	arModbusOdczytCykliczny[intPetlaPierwszySkan].bAdresUrzadzenia := bAdres;
	arModbusOdczytCykliczny[intPetlaPierwszySkan].bFunkcja := TO_BYTE(enumModbusKodyFunkcji.OdczytNRejestrow);
	arModbusOdczytCykliczny[intPetlaPierwszySkan].uiAdresRejestru := 50544;
	arModbusOdczytCykliczny[intPetlaPierwszySkan].ltCzestotliwosc := TIME_TO_LTIME(tMinimalnyCzasRaportowania);
	arModbusOdczytCykliczny[intPetlaPierwszySkan].pZmiennaReferencyjna := ADR(wMocCzynnaL1Hi);
	intPetlaPierwszySkan := intPetlaPierwszySkan + 1;
	
	arModbusOdczytCykliczny[intPetlaPierwszySkan].bAdresUrzadzenia := bAdres;
	arModbusOdczytCykliczny[intPetlaPierwszySkan].bFunkcja := TO_BYTE(enumModbusKodyFunkcji.OdczytNRejestrow);
	arModbusOdczytCykliczny[intPetlaPierwszySkan].uiAdresRejestru := 50545;
	arModbusOdczytCykliczny[intPetlaPierwszySkan].ltCzestotliwosc := TIME_TO_LTIME(tMinimalnyCzasRaportowania);
	arModbusOdczytCykliczny[intPetlaPierwszySkan].pZmiennaReferencyjna := ADR(wMocCzynnaL1Lo);
	intPetlaPierwszySkan := intPetlaPierwszySkan + 1;
	
	arModbusOdczytCykliczny[intPetlaPierwszySkan].bAdresUrzadzenia := bAdres;
	arModbusOdczytCykliczny[intPetlaPierwszySkan].bFunkcja := TO_BYTE(enumModbusKodyFunkcji.OdczytNRejestrow);
	arModbusOdczytCykliczny[intPetlaPierwszySkan].uiAdresRejestru := 50546;
	arModbusOdczytCykliczny[intPetlaPierwszySkan].ltCzestotliwosc := TIME_TO_LTIME(tMinimalnyCzasRaportowania);
	arModbusOdczytCykliczny[intPetlaPierwszySkan].pZmiennaReferencyjna := ADR(wMocCzynnaL2Hi);
	intPetlaPierwszySkan := intPetlaPierwszySkan + 1;
	
	arModbusOdczytCykliczny[intPetlaPierwszySkan].bAdresUrzadzenia := bAdres;
	arModbusOdczytCykliczny[intPetlaPierwszySkan].bFunkcja := TO_BYTE(enumModbusKodyFunkcji.OdczytNRejestrow);
	arModbusOdczytCykliczny[intPetlaPierwszySkan].uiAdresRejestru := 50547;
	arModbusOdczytCykliczny[intPetlaPierwszySkan].ltCzestotliwosc := TIME_TO_LTIME(tMinimalnyCzasRaportowania);
	arModbusOdczytCykliczny[intPetlaPierwszySkan].pZmiennaReferencyjna := ADR(wMocCzynnaL2Lo);
	intPetlaPierwszySkan := intPetlaPierwszySkan + 1;
	
	arModbusOdczytCykliczny[intPetlaPierwszySkan].bAdresUrzadzenia := bAdres;
	arModbusOdczytCykliczny[intPetlaPierwszySkan].bFunkcja := TO_BYTE(enumModbusKodyFunkcji.OdczytNRejestrow);
	arModbusOdczytCykliczny[intPetlaPierwszySkan].uiAdresRejestru := 50548;
	arModbusOdczytCykliczny[intPetlaPierwszySkan].ltCzestotliwosc := TIME_TO_LTIME(tMinimalnyCzasRaportowania);
	arModbusOdczytCykliczny[intPetlaPierwszySkan].pZmiennaReferencyjna := ADR(wMocCzynnaL3Hi);
	intPetlaPierwszySkan := intPetlaPierwszySkan + 1;
	
	arModbusOdczytCykliczny[intPetlaPierwszySkan].bAdresUrzadzenia := bAdres;
	arModbusOdczytCykliczny[intPetlaPierwszySkan].bFunkcja := TO_BYTE(enumModbusKodyFunkcji.OdczytNRejestrow);
	arModbusOdczytCykliczny[intPetlaPierwszySkan].uiAdresRejestru := 50549;
	arModbusOdczytCykliczny[intPetlaPierwszySkan].ltCzestotliwosc := TIME_TO_LTIME(tMinimalnyCzasRaportowania);
	arModbusOdczytCykliczny[intPetlaPierwszySkan].pZmiennaReferencyjna := ADR(wMocCzynnaL3Lo);
	intPetlaPierwszySkan := intPetlaPierwszySkan + 1;	
	
	arModbusOdczytCykliczny[intPetlaPierwszySkan].bAdresUrzadzenia := bAdres;
	arModbusOdczytCykliczny[intPetlaPierwszySkan].bFunkcja := TO_BYTE(enumModbusKodyFunkcji.OdczytNRejestrow);
	arModbusOdczytCykliczny[intPetlaPierwszySkan].uiAdresRejestru := 50556;
	arModbusOdczytCykliczny[intPetlaPierwszySkan].ltCzestotliwosc := TIME_TO_LTIME(tMinimalnyCzasRaportowania);
	arModbusOdczytCykliczny[intPetlaPierwszySkan].pZmiennaReferencyjna := ADR(wMocPozornaL1Hi);
	intPetlaPierwszySkan := intPetlaPierwszySkan + 1;

	arModbusOdczytCykliczny[intPetlaPierwszySkan].bAdresUrzadzenia := bAdres;
	arModbusOdczytCykliczny[intPetlaPierwszySkan].bFunkcja := TO_BYTE(enumModbusKodyFunkcji.OdczytNRejestrow);
	arModbusOdczytCykliczny[intPetlaPierwszySkan].uiAdresRejestru := 50557;
	arModbusOdczytCykliczny[intPetlaPierwszySkan].ltCzestotliwosc := TIME_TO_LTIME(tMinimalnyCzasRaportowania);
	arModbusOdczytCykliczny[intPetlaPierwszySkan].pZmiennaReferencyjna := ADR(wMocPozornaL1Lo);
	intPetlaPierwszySkan := intPetlaPierwszySkan + 1;	

	arModbusOdczytCykliczny[intPetlaPierwszySkan].bAdresUrzadzenia := bAdres;
	arModbusOdczytCykliczny[intPetlaPierwszySkan].bFunkcja := TO_BYTE(enumModbusKodyFunkcji.OdczytNRejestrow);
	arModbusOdczytCykliczny[intPetlaPierwszySkan].uiAdresRejestru := 50558;
	arModbusOdczytCykliczny[intPetlaPierwszySkan].ltCzestotliwosc := TIME_TO_LTIME(tMinimalnyCzasRaportowania);
	arModbusOdczytCykliczny[intPetlaPierwszySkan].pZmiennaReferencyjna := ADR(wMocPozornaL2Hi);
	intPetlaPierwszySkan := intPetlaPierwszySkan + 1;

	arModbusOdczytCykliczny[intPetlaPierwszySkan].bAdresUrzadzenia := bAdres;
	arModbusOdczytCykliczny[intPetlaPierwszySkan].bFunkcja := TO_BYTE(enumModbusKodyFunkcji.OdczytNRejestrow);
	arModbusOdczytCykliczny[intPetlaPierwszySkan].uiAdresRejestru := 50559;
	arModbusOdczytCykliczny[intPetlaPierwszySkan].ltCzestotliwosc := TIME_TO_LTIME(tMinimalnyCzasRaportowania);
	arModbusOdczytCykliczny[intPetlaPierwszySkan].pZmiennaReferencyjna := ADR(wMocPozornaL2Lo);
	intPetlaPierwszySkan := intPetlaPierwszySkan + 1;	

	arModbusOdczytCykliczny[intPetlaPierwszySkan].bAdresUrzadzenia := bAdres;
	arModbusOdczytCykliczny[intPetlaPierwszySkan].bFunkcja := TO_BYTE(enumModbusKodyFunkcji.OdczytNRejestrow);
	arModbusOdczytCykliczny[intPetlaPierwszySkan].uiAdresRejestru := 50560;
	arModbusOdczytCykliczny[intPetlaPierwszySkan].ltCzestotliwosc := TIME_TO_LTIME(tMinimalnyCzasRaportowania);
	arModbusOdczytCykliczny[intPetlaPierwszySkan].pZmiennaReferencyjna := ADR(wMocPozornaL3Hi);
	intPetlaPierwszySkan := intPetlaPierwszySkan + 1;

	arModbusOdczytCykliczny[intPetlaPierwszySkan].bAdresUrzadzenia := bAdres;
	arModbusOdczytCykliczny[intPetlaPierwszySkan].bFunkcja := TO_BYTE(enumModbusKodyFunkcji.OdczytNRejestrow);
	arModbusOdczytCykliczny[intPetlaPierwszySkan].uiAdresRejestru := 50561;
	arModbusOdczytCykliczny[intPetlaPierwszySkan].ltCzestotliwosc := TIME_TO_LTIME(tMinimalnyCzasRaportowania);
	arModbusOdczytCykliczny[intPetlaPierwszySkan].pZmiennaReferencyjna := ADR(wMocPozornaL3Lo);
	intPetlaPierwszySkan := intPetlaPierwszySkan + 1;	
	
	arModbusOdczytCykliczny[intPetlaPierwszySkan].bAdresUrzadzenia := bAdres;
	arModbusOdczytCykliczny[intPetlaPierwszySkan].bFunkcja := TO_BYTE(enumModbusKodyFunkcji.OdczytNRejestrow);
	arModbusOdczytCykliczny[intPetlaPierwszySkan].uiAdresRejestru := 50562;
	arModbusOdczytCykliczny[intPetlaPierwszySkan].ltCzestotliwosc := TIME_TO_LTIME(tMinimalnyCzasRaportowania);
	arModbusOdczytCykliczny[intPetlaPierwszySkan].pZmiennaReferencyjna := ADR(wWspolczynnikMocyL1Hi);
	intPetlaPierwszySkan := intPetlaPierwszySkan + 1;

	arModbusOdczytCykliczny[intPetlaPierwszySkan].bAdresUrzadzenia := bAdres;
	arModbusOdczytCykliczny[intPetlaPierwszySkan].bFunkcja := TO_BYTE(enumModbusKodyFunkcji.OdczytNRejestrow);
	arModbusOdczytCykliczny[intPetlaPierwszySkan].uiAdresRejestru := 50563;
	arModbusOdczytCykliczny[intPetlaPierwszySkan].ltCzestotliwosc := TIME_TO_LTIME(tMinimalnyCzasRaportowania);
	arModbusOdczytCykliczny[intPetlaPierwszySkan].pZmiennaReferencyjna := ADR(wWspolczynnikMocyL1Lo);
	intPetlaPierwszySkan := intPetlaPierwszySkan + 1;
	
	arModbusOdczytCykliczny[intPetlaPierwszySkan].bAdresUrzadzenia := bAdres;
	arModbusOdczytCykliczny[intPetlaPierwszySkan].bFunkcja := TO_BYTE(enumModbusKodyFunkcji.OdczytNRejestrow);
	arModbusOdczytCykliczny[intPetlaPierwszySkan].uiAdresRejestru := 50564;
	arModbusOdczytCykliczny[intPetlaPierwszySkan].ltCzestotliwosc := TIME_TO_LTIME(tMinimalnyCzasRaportowania);
	arModbusOdczytCykliczny[intPetlaPierwszySkan].pZmiennaReferencyjna := ADR(wWspolczynnikMocyL2Hi);
	intPetlaPierwszySkan := intPetlaPierwszySkan + 1;

	arModbusOdczytCykliczny[intPetlaPierwszySkan].bAdresUrzadzenia := bAdres;
	arModbusOdczytCykliczny[intPetlaPierwszySkan].bFunkcja := TO_BYTE(enumModbusKodyFunkcji.OdczytNRejestrow);
	arModbusOdczytCykliczny[intPetlaPierwszySkan].uiAdresRejestru := 50565;
	arModbusOdczytCykliczny[intPetlaPierwszySkan].ltCzestotliwosc := TIME_TO_LTIME(tMinimalnyCzasRaportowania);
	arModbusOdczytCykliczny[intPetlaPierwszySkan].pZmiennaReferencyjna := ADR(wWspolczynnikMocyL2Lo);
	intPetlaPierwszySkan := intPetlaPierwszySkan + 1;
	
	arModbusOdczytCykliczny[intPetlaPierwszySkan].bAdresUrzadzenia := bAdres;
	arModbusOdczytCykliczny[intPetlaPierwszySkan].bFunkcja := TO_BYTE(enumModbusKodyFunkcji.OdczytNRejestrow);
	arModbusOdczytCykliczny[intPetlaPierwszySkan].uiAdresRejestru := 50566;
	arModbusOdczytCykliczny[intPetlaPierwszySkan].ltCzestotliwosc := TIME_TO_LTIME(tMinimalnyCzasRaportowania);
	arModbusOdczytCykliczny[intPetlaPierwszySkan].pZmiennaReferencyjna := ADR(wWspolczynnikMocyL3Hi);
	intPetlaPierwszySkan := intPetlaPierwszySkan + 1;

	arModbusOdczytCykliczny[intPetlaPierwszySkan].bAdresUrzadzenia := bAdres;
	arModbusOdczytCykliczny[intPetlaPierwszySkan].bFunkcja := TO_BYTE(enumModbusKodyFunkcji.OdczytNRejestrow);
	arModbusOdczytCykliczny[intPetlaPierwszySkan].uiAdresRejestru := 50567;
	arModbusOdczytCykliczny[intPetlaPierwszySkan].ltCzestotliwosc := TIME_TO_LTIME(tMinimalnyCzasRaportowania);
	arModbusOdczytCykliczny[intPetlaPierwszySkan].pZmiennaReferencyjna := ADR(wWspolczynnikMocyL3Lo);
	intPetlaPierwszySkan := intPetlaPierwszySkan + 1;
	
	arModbusOdczytCykliczny[intPetlaPierwszySkan].bAdresUrzadzenia := bAdres;
	arModbusOdczytCykliczny[intPetlaPierwszySkan].bFunkcja := TO_BYTE(enumModbusKodyFunkcji.OdczytNRejestrow);
	arModbusOdczytCykliczny[intPetlaPierwszySkan].uiAdresRejestru := 856;
	arModbusOdczytCykliczny[intPetlaPierwszySkan].ltCzestotliwosc := TIME_TO_LTIME(tMinimalnyCzasRaportowania);
	arModbusOdczytCykliczny[intPetlaPierwszySkan].pZmiennaReferencyjna := ADR(wEnergiaCzynnaPobranaHi);
	intPetlaPierwszySkan := intPetlaPierwszySkan + 1;

	arModbusOdczytCykliczny[intPetlaPierwszySkan].bAdresUrzadzenia := bAdres;
	arModbusOdczytCykliczny[intPetlaPierwszySkan].bFunkcja := TO_BYTE(enumModbusKodyFunkcji.OdczytNRejestrow);
	arModbusOdczytCykliczny[intPetlaPierwszySkan].uiAdresRejestru := 857;
	arModbusOdczytCykliczny[intPetlaPierwszySkan].ltCzestotliwosc := TIME_TO_LTIME(tMinimalnyCzasRaportowania);
	arModbusOdczytCykliczny[intPetlaPierwszySkan].pZmiennaReferencyjna := ADR(wEnergiaCzynnaPobranaLo);
	intPetlaPierwszySkan := intPetlaPierwszySkan + 1;
	
	arModbusOdczytCykliczny[intPetlaPierwszySkan].bAdresUrzadzenia := bAdres;
	arModbusOdczytCykliczny[intPetlaPierwszySkan].bFunkcja := TO_BYTE(enumModbusKodyFunkcji.OdczytNRejestrow);
	arModbusOdczytCykliczny[intPetlaPierwszySkan].uiAdresRejestru := 858;
	arModbusOdczytCykliczny[intPetlaPierwszySkan].ltCzestotliwosc := TIME_TO_LTIME(tMinimalnyCzasRaportowania);
	arModbusOdczytCykliczny[intPetlaPierwszySkan].pZmiennaReferencyjna := ADR(wEnergiaBiernaPobranaHi);
	intPetlaPierwszySkan := intPetlaPierwszySkan + 1;

	arModbusOdczytCykliczny[intPetlaPierwszySkan].bAdresUrzadzenia := bAdres;
	arModbusOdczytCykliczny[intPetlaPierwszySkan].bFunkcja := TO_BYTE(enumModbusKodyFunkcji.OdczytNRejestrow);
	arModbusOdczytCykliczny[intPetlaPierwszySkan].uiAdresRejestru := 859;
	arModbusOdczytCykliczny[intPetlaPierwszySkan].ltCzestotliwosc := TIME_TO_LTIME(tMinimalnyCzasRaportowania);
	arModbusOdczytCykliczny[intPetlaPierwszySkan].pZmiennaReferencyjna := ADR(wEnergiaBiernaPobranaLo);
	intPetlaPierwszySkan := intPetlaPierwszySkan + 1;
	
	arModbusOdczytCykliczny[intPetlaPierwszySkan].bAdresUrzadzenia := bAdres;
	arModbusOdczytCykliczny[intPetlaPierwszySkan].bFunkcja := TO_BYTE(enumModbusKodyFunkcji.OdczytNRejestrow);
	arModbusOdczytCykliczny[intPetlaPierwszySkan].uiAdresRejestru := 860;
	arModbusOdczytCykliczny[intPetlaPierwszySkan].ltCzestotliwosc := TIME_TO_LTIME(tMinimalnyCzasRaportowania);
	arModbusOdczytCykliczny[intPetlaPierwszySkan].pZmiennaReferencyjna := ADR(wEnergiaPozornaPobranaHi);
	intPetlaPierwszySkan := intPetlaPierwszySkan + 1;

	arModbusOdczytCykliczny[intPetlaPierwszySkan].bAdresUrzadzenia := bAdres;
	arModbusOdczytCykliczny[intPetlaPierwszySkan].bFunkcja := TO_BYTE(enumModbusKodyFunkcji.OdczytNRejestrow);
	arModbusOdczytCykliczny[intPetlaPierwszySkan].uiAdresRejestru := 861;
	arModbusOdczytCykliczny[intPetlaPierwszySkan].ltCzestotliwosc := TIME_TO_LTIME(tMinimalnyCzasRaportowania);
	arModbusOdczytCykliczny[intPetlaPierwszySkan].pZmiennaReferencyjna := ADR(wEnergiaPozornaPobranaLo);
	intPetlaPierwszySkan := intPetlaPierwszySkan + 1;
	
	arModbusOdczytCykliczny[intPetlaPierwszySkan].bAdresUrzadzenia := bAdres;
	arModbusOdczytCykliczny[intPetlaPierwszySkan].bFunkcja := TO_BYTE(enumModbusKodyFunkcji.OdczytNRejestrow);
	arModbusOdczytCykliczny[intPetlaPierwszySkan].uiAdresRejestru := 51038;
	arModbusOdczytCykliczny[intPetlaPierwszySkan].ltCzestotliwosc := TIME_TO_LTIME(tMinimalnyCzasRaportowania);
	arModbusOdczytCykliczny[intPetlaPierwszySkan].pZmiennaReferencyjna := ADR(wPradSredniL1Hi);
	intPetlaPierwszySkan := intPetlaPierwszySkan + 1;

	arModbusOdczytCykliczny[intPetlaPierwszySkan].bAdresUrzadzenia := bAdres;
	arModbusOdczytCykliczny[intPetlaPierwszySkan].bFunkcja := TO_BYTE(enumModbusKodyFunkcji.OdczytNRejestrow);
	arModbusOdczytCykliczny[intPetlaPierwszySkan].uiAdresRejestru := 51039;
	arModbusOdczytCykliczny[intPetlaPierwszySkan].ltCzestotliwosc := TIME_TO_LTIME(tMinimalnyCzasRaportowania);
	arModbusOdczytCykliczny[intPetlaPierwszySkan].pZmiennaReferencyjna := ADR(wPradSredniL1Lo);
	intPetlaPierwszySkan := intPetlaPierwszySkan + 1;
	
	arModbusOdczytCykliczny[intPetlaPierwszySkan].bAdresUrzadzenia := bAdres;
	arModbusOdczytCykliczny[intPetlaPierwszySkan].bFunkcja := TO_BYTE(enumModbusKodyFunkcji.OdczytNRejestrow);
	arModbusOdczytCykliczny[intPetlaPierwszySkan].uiAdresRejestru := 51040;
	arModbusOdczytCykliczny[intPetlaPierwszySkan].ltCzestotliwosc := TIME_TO_LTIME(tMinimalnyCzasRaportowania);
	arModbusOdczytCykliczny[intPetlaPierwszySkan].pZmiennaReferencyjna := ADR(wPradSredniL2Hi);
	intPetlaPierwszySkan := intPetlaPierwszySkan + 1;

	arModbusOdczytCykliczny[intPetlaPierwszySkan].bAdresUrzadzenia := bAdres;
	arModbusOdczytCykliczny[intPetlaPierwszySkan].bFunkcja := TO_BYTE(enumModbusKodyFunkcji.OdczytNRejestrow);
	arModbusOdczytCykliczny[intPetlaPierwszySkan].uiAdresRejestru := 51041;
	arModbusOdczytCykliczny[intPetlaPierwszySkan].ltCzestotliwosc := TIME_TO_LTIME(tMinimalnyCzasRaportowania);
	arModbusOdczytCykliczny[intPetlaPierwszySkan].pZmiennaReferencyjna := ADR(wPradSredniL2Lo);
	intPetlaPierwszySkan := intPetlaPierwszySkan + 1;
	
	arModbusOdczytCykliczny[intPetlaPierwszySkan].bAdresUrzadzenia := bAdres;
	arModbusOdczytCykliczny[intPetlaPierwszySkan].bFunkcja := TO_BYTE(enumModbusKodyFunkcji.OdczytNRejestrow);
	arModbusOdczytCykliczny[intPetlaPierwszySkan].uiAdresRejestru := 51042;
	arModbusOdczytCykliczny[intPetlaPierwszySkan].ltCzestotliwosc := TIME_TO_LTIME(tMinimalnyCzasRaportowania);
	arModbusOdczytCykliczny[intPetlaPierwszySkan].pZmiennaReferencyjna := ADR(wPradSredniL3Hi);
	intPetlaPierwszySkan := intPetlaPierwszySkan + 1;

	arModbusOdczytCykliczny[intPetlaPierwszySkan].bAdresUrzadzenia := bAdres;
	arModbusOdczytCykliczny[intPetlaPierwszySkan].bFunkcja := TO_BYTE(enumModbusKodyFunkcji.OdczytNRejestrow);
	arModbusOdczytCykliczny[intPetlaPierwszySkan].uiAdresRejestru := 51043;
	arModbusOdczytCykliczny[intPetlaPierwszySkan].ltCzestotliwosc := TIME_TO_LTIME(tMinimalnyCzasRaportowania);
	arModbusOdczytCykliczny[intPetlaPierwszySkan].pZmiennaReferencyjna := ADR(wPradSredniL3Lo);
	intPetlaPierwszySkan := intPetlaPierwszySkan + 1;

	arModbusOdczytCykliczny[intPetlaPierwszySkan].bAdresUrzadzenia := bAdres;
	arModbusOdczytCykliczny[intPetlaPierwszySkan].bFunkcja := TO_BYTE(enumModbusKodyFunkcji.OdczytNRejestrow);
	arModbusOdczytCykliczny[intPetlaPierwszySkan].uiAdresRejestru := 51046;
	arModbusOdczytCykliczny[intPetlaPierwszySkan].ltCzestotliwosc := TIME_TO_LTIME(tMinimalnyCzasRaportowania);
	arModbusOdczytCykliczny[intPetlaPierwszySkan].pZmiennaReferencyjna := ADR(wMocCzynnaSredniaHi);
	intPetlaPierwszySkan := intPetlaPierwszySkan + 1;

	arModbusOdczytCykliczny[intPetlaPierwszySkan].bAdresUrzadzenia := bAdres;
	arModbusOdczytCykliczny[intPetlaPierwszySkan].bFunkcja := TO_BYTE(enumModbusKodyFunkcji.OdczytNRejestrow);
	arModbusOdczytCykliczny[intPetlaPierwszySkan].uiAdresRejestru := 51047;
	arModbusOdczytCykliczny[intPetlaPierwszySkan].ltCzestotliwosc := TIME_TO_LTIME(tMinimalnyCzasRaportowania);
	arModbusOdczytCykliczny[intPetlaPierwszySkan].pZmiennaReferencyjna := ADR(wMocCzynnaSredniaLo);
	intPetlaPierwszySkan := intPetlaPierwszySkan + 1;

	arModbusOdczytCykliczny[intPetlaPierwszySkan].bAdresUrzadzenia := bAdres;
	arModbusOdczytCykliczny[intPetlaPierwszySkan].bFunkcja := TO_BYTE(enumModbusKodyFunkcji.OdczytNRejestrow);
	arModbusOdczytCykliczny[intPetlaPierwszySkan].uiAdresRejestru := 51052;
	arModbusOdczytCykliczny[intPetlaPierwszySkan].ltCzestotliwosc := TIME_TO_LTIME(tMinimalnyCzasRaportowania);
	arModbusOdczytCykliczny[intPetlaPierwszySkan].pZmiennaReferencyjna := ADR(wMocBiernaSredniaHi);
	intPetlaPierwszySkan := intPetlaPierwszySkan + 1;

	arModbusOdczytCykliczny[intPetlaPierwszySkan].bAdresUrzadzenia := bAdres;
	arModbusOdczytCykliczny[intPetlaPierwszySkan].bFunkcja := TO_BYTE(enumModbusKodyFunkcji.OdczytNRejestrow);
	arModbusOdczytCykliczny[intPetlaPierwszySkan].uiAdresRejestru := 51053;
	arModbusOdczytCykliczny[intPetlaPierwszySkan].ltCzestotliwosc := TIME_TO_LTIME(tMinimalnyCzasRaportowania);
	arModbusOdczytCykliczny[intPetlaPierwszySkan].pZmiennaReferencyjna := ADR(wMocBiernaSredniaLo);
	intPetlaPierwszySkan := intPetlaPierwszySkan + 1;

	arModbusOdczytCykliczny[intPetlaPierwszySkan].bAdresUrzadzenia := bAdres;
	arModbusOdczytCykliczny[intPetlaPierwszySkan].bFunkcja := TO_BYTE(enumModbusKodyFunkcji.OdczytNRejestrow);
	arModbusOdczytCykliczny[intPetlaPierwszySkan].uiAdresRejestru := 51054;
	arModbusOdczytCykliczny[intPetlaPierwszySkan].ltCzestotliwosc := TIME_TO_LTIME(tMinimalnyCzasRaportowania);
	arModbusOdczytCykliczny[intPetlaPierwszySkan].pZmiennaReferencyjna := ADR(wMocPozornaSredniaHi);
	intPetlaPierwszySkan := intPetlaPierwszySkan + 1;

	arModbusOdczytCykliczny[intPetlaPierwszySkan].bAdresUrzadzenia := bAdres;
	arModbusOdczytCykliczny[intPetlaPierwszySkan].bFunkcja := TO_BYTE(enumModbusKodyFunkcji.OdczytNRejestrow);
	arModbusOdczytCykliczny[intPetlaPierwszySkan].uiAdresRejestru := 51055;
	arModbusOdczytCykliczny[intPetlaPierwszySkan].ltCzestotliwosc := TIME_TO_LTIME(tMinimalnyCzasRaportowania);
	arModbusOdczytCykliczny[intPetlaPierwszySkan].pZmiennaReferencyjna := ADR(wMocPozornaSredniaLo);
	intPetlaPierwszySkan := intPetlaPierwszySkan + 1;

	arModbusOdczytCykliczny[intPetlaPierwszySkan].bAdresUrzadzenia := bAdres;
	arModbusOdczytCykliczny[intPetlaPierwszySkan].bFunkcja := TO_BYTE(enumModbusKodyFunkcji.OdczytNRejestrow);
	arModbusOdczytCykliczny[intPetlaPierwszySkan].uiAdresRejestru := 51062;
	arModbusOdczytCykliczny[intPetlaPierwszySkan].ltCzestotliwosc := TIME_TO_LTIME(tMinimalnyCzasRaportowania);
	arModbusOdczytCykliczny[intPetlaPierwszySkan].pZmiennaReferencyjna := ADR(wMaksymalneNapiecieL1Hi);
	intPetlaPierwszySkan := intPetlaPierwszySkan + 1;

	arModbusOdczytCykliczny[intPetlaPierwszySkan].bAdresUrzadzenia := bAdres;
	arModbusOdczytCykliczny[intPetlaPierwszySkan].bFunkcja := TO_BYTE(enumModbusKodyFunkcji.OdczytNRejestrow);
	arModbusOdczytCykliczny[intPetlaPierwszySkan].uiAdresRejestru := 51063;
	arModbusOdczytCykliczny[intPetlaPierwszySkan].ltCzestotliwosc := TIME_TO_LTIME(tMinimalnyCzasRaportowania);
	arModbusOdczytCykliczny[intPetlaPierwszySkan].pZmiennaReferencyjna := ADR(wMaksymalneNapiecieL1Lo);
	intPetlaPierwszySkan := intPetlaPierwszySkan + 1;

	arModbusOdczytCykliczny[intPetlaPierwszySkan].bAdresUrzadzenia := bAdres;
	arModbusOdczytCykliczny[intPetlaPierwszySkan].bFunkcja := TO_BYTE(enumModbusKodyFunkcji.OdczytNRejestrow);
	arModbusOdczytCykliczny[intPetlaPierwszySkan].uiAdresRejestru := 51064;
	arModbusOdczytCykliczny[intPetlaPierwszySkan].ltCzestotliwosc := TIME_TO_LTIME(tMinimalnyCzasRaportowania);
	arModbusOdczytCykliczny[intPetlaPierwszySkan].pZmiennaReferencyjna := ADR(wMaksymalneNapiecieL2Hi);
	intPetlaPierwszySkan := intPetlaPierwszySkan + 1;

	arModbusOdczytCykliczny[intPetlaPierwszySkan].bAdresUrzadzenia := bAdres;
	arModbusOdczytCykliczny[intPetlaPierwszySkan].bFunkcja := TO_BYTE(enumModbusKodyFunkcji.OdczytNRejestrow);
	arModbusOdczytCykliczny[intPetlaPierwszySkan].uiAdresRejestru := 51065;
	arModbusOdczytCykliczny[intPetlaPierwszySkan].ltCzestotliwosc := TIME_TO_LTIME(tMinimalnyCzasRaportowania);
	arModbusOdczytCykliczny[intPetlaPierwszySkan].pZmiennaReferencyjna := ADR(wMaksymalneNapiecieL2Lo);
	intPetlaPierwszySkan := intPetlaPierwszySkan + 1;

	arModbusOdczytCykliczny[intPetlaPierwszySkan].bAdresUrzadzenia := bAdres;
	arModbusOdczytCykliczny[intPetlaPierwszySkan].bFunkcja := TO_BYTE(enumModbusKodyFunkcji.OdczytNRejestrow);
	arModbusOdczytCykliczny[intPetlaPierwszySkan].uiAdresRejestru := 51066;
	arModbusOdczytCykliczny[intPetlaPierwszySkan].ltCzestotliwosc := TIME_TO_LTIME(tMinimalnyCzasRaportowania);
	arModbusOdczytCykliczny[intPetlaPierwszySkan].pZmiennaReferencyjna := ADR(wMaksymalneNapiecieL3Hi);
	intPetlaPierwszySkan := intPetlaPierwszySkan + 1;

	arModbusOdczytCykliczny[intPetlaPierwszySkan].bAdresUrzadzenia := bAdres;
	arModbusOdczytCykliczny[intPetlaPierwszySkan].bFunkcja := TO_BYTE(enumModbusKodyFunkcji.OdczytNRejestrow);
	arModbusOdczytCykliczny[intPetlaPierwszySkan].uiAdresRejestru := 51067;
	arModbusOdczytCykliczny[intPetlaPierwszySkan].ltCzestotliwosc := TIME_TO_LTIME(tMinimalnyCzasRaportowania);
	arModbusOdczytCykliczny[intPetlaPierwszySkan].pZmiennaReferencyjna := ADR(wMaksymalneNapiecieL3Lo);
	intPetlaPierwszySkan := intPetlaPierwszySkan + 1;

	arModbusOdczytCykliczny[intPetlaPierwszySkan].bAdresUrzadzenia := bAdres;
	arModbusOdczytCykliczny[intPetlaPierwszySkan].bFunkcja := TO_BYTE(enumModbusKodyFunkcji.OdczytNRejestrow);
	arModbusOdczytCykliczny[intPetlaPierwszySkan].uiAdresRejestru := 51539;
	arModbusOdczytCykliczny[intPetlaPierwszySkan].ltCzestotliwosc := TIME_TO_LTIME(tMinimalnyCzasRaportowania);
	arModbusOdczytCykliczny[intPetlaPierwszySkan].pZmiennaReferencyjna := ADR(wTHDNapieciaL1);
	intPetlaPierwszySkan := intPetlaPierwszySkan + 1;

	arModbusOdczytCykliczny[intPetlaPierwszySkan].bAdresUrzadzenia := bAdres;
	arModbusOdczytCykliczny[intPetlaPierwszySkan].bFunkcja := TO_BYTE(enumModbusKodyFunkcji.OdczytNRejestrow);
	arModbusOdczytCykliczny[intPetlaPierwszySkan].uiAdresRejestru := 51540;
	arModbusOdczytCykliczny[intPetlaPierwszySkan].ltCzestotliwosc := TIME_TO_LTIME(tMinimalnyCzasRaportowania);
	arModbusOdczytCykliczny[intPetlaPierwszySkan].pZmiennaReferencyjna := ADR(wTHDNapieciaL2);
	intPetlaPierwszySkan := intPetlaPierwszySkan + 1;

	arModbusOdczytCykliczny[intPetlaPierwszySkan].bAdresUrzadzenia := bAdres;
	arModbusOdczytCykliczny[intPetlaPierwszySkan].bFunkcja := TO_BYTE(enumModbusKodyFunkcji.OdczytNRejestrow);
	arModbusOdczytCykliczny[intPetlaPierwszySkan].uiAdresRejestru := 51541;
	arModbusOdczytCykliczny[intPetlaPierwszySkan].ltCzestotliwosc := TIME_TO_LTIME(tMinimalnyCzasRaportowania);
	arModbusOdczytCykliczny[intPetlaPierwszySkan].pZmiennaReferencyjna := ADR(wTHDNapieciaL3);
	intPetlaPierwszySkan := intPetlaPierwszySkan + 1;

	arModbusOdczytCykliczny[intPetlaPierwszySkan].bAdresUrzadzenia := bAdres;
	arModbusOdczytCykliczny[intPetlaPierwszySkan].bFunkcja := TO_BYTE(enumModbusKodyFunkcji.OdczytNRejestrow);
	arModbusOdczytCykliczny[intPetlaPierwszySkan].uiAdresRejestru := 51542;
	arModbusOdczytCykliczny[intPetlaPierwszySkan].ltCzestotliwosc := TIME_TO_LTIME(tMinimalnyCzasRaportowania);
	arModbusOdczytCykliczny[intPetlaPierwszySkan].pZmiennaReferencyjna := ADR(wTHDPraduL1);
	intPetlaPierwszySkan := intPetlaPierwszySkan + 1;

	arModbusOdczytCykliczny[intPetlaPierwszySkan].bAdresUrzadzenia := bAdres;
	arModbusOdczytCykliczny[intPetlaPierwszySkan].bFunkcja := TO_BYTE(enumModbusKodyFunkcji.OdczytNRejestrow);
	arModbusOdczytCykliczny[intPetlaPierwszySkan].uiAdresRejestru := 51543;
	arModbusOdczytCykliczny[intPetlaPierwszySkan].ltCzestotliwosc := TIME_TO_LTIME(tMinimalnyCzasRaportowania);
	arModbusOdczytCykliczny[intPetlaPierwszySkan].pZmiennaReferencyjna := ADR(wTHDPraduL2);
	intPetlaPierwszySkan := intPetlaPierwszySkan + 1;

	arModbusOdczytCykliczny[intPetlaPierwszySkan].bAdresUrzadzenia := bAdres;
	arModbusOdczytCykliczny[intPetlaPierwszySkan].bFunkcja := TO_BYTE(enumModbusKodyFunkcji.OdczytNRejestrow);
	arModbusOdczytCykliczny[intPetlaPierwszySkan].uiAdresRejestru := 51544;
	arModbusOdczytCykliczny[intPetlaPierwszySkan].ltCzestotliwosc := TIME_TO_LTIME(tMinimalnyCzasRaportowania);
	arModbusOdczytCykliczny[intPetlaPierwszySkan].pZmiennaReferencyjna := ADR(wTHDPraduL3);
	intPetlaPierwszySkan := intPetlaPierwszySkan + 1;
END_IF

//obsluga komunikatu przychodzacego z IZE

IF 	sKomunikat <> sKomunikatPamiec AND xPoInicjalizacji THEN
	sKomunikatPamiec := sKomunikat;
	IF fnIDOdbiorcyMatch(sKomunikat , sIdInstancji) THEN
		sDane := '';
		//zapytanie typu Q
		IF fnKomunikatTyp(sKomunikat) = 'Q' AND arModbusStatusKomunikacji[bAdres] = enumModbusStatus.KomunikacjaPrawidlowa THEN
			//Napięcia fazowe
			IF fnKomunikatDaneSzukajWartosci(sKomunikat , 'VOLTL1=') = '?' OR fnKomunikatDaneSzukajWartosci(sKomunikat , 'ALL=') = '?' THEN
				fnKomunikatDaneDodaj_xOverFlow(sDane := sDane , sAtrybut := 'VOLTL1=' , sWartosc := REAL_TO_STRING(rNapiecieL1) , xOverFlow := xOverFlow);
				IF xOverFlow = TRUE THEN
					fnZapiszKomunikat(	sCalyKomunikat := '' ,
								sTypKomunikatu := 'A' ,
								sMnemonik := sMnemonik ,
								sMACAdres := sMACAdres ,
								sIDNadawcy := sIdInstancji ,
								sIDOdbiorcy := sIdAplikacji ,
								sDaneZapasowe := sDaneZapasowe ,
								sDane := sDane ,
								arTablicaKomunikatow := arTablicaKomunikatow ,
								intTablicaKomunikatowZnacznikZapisu := intTablicaKomunikatowZnacznikZapisu ,
								intTablicaKomunikatowRozmiar := intTablicaKomunikatowRozmiar ,
								sWyslanyKomunikat := sWyslanyKomunikatDummy);
					sDane := '';
				END_IF
			END_IF
			IF fnKomunikatDaneSzukajWartosci(sKomunikat , 'VOLTL2=') = '?' OR fnKomunikatDaneSzukajWartosci(sKomunikat , 'ALL=') = '?' THEN
				fnKomunikatDaneDodaj_xOverFlow(sDane := sDane , sAtrybut := 'VOLTL2=' , sWartosc := REAL_TO_STRING(rNapiecieL2) , xOverFlow := xOverFlow);
				IF xOverFlow = TRUE THEN
					fnZapiszKomunikat(	sCalyKomunikat := '' ,
								sTypKomunikatu := 'A' ,
								sMnemonik := sMnemonik ,
								sMACAdres := sMACAdres ,
								sIDNadawcy := sIdInstancji ,
								sIDOdbiorcy := sIdAplikacji ,
								sDaneZapasowe := sDaneZapasowe ,
								sDane := sDane ,
								arTablicaKomunikatow := arTablicaKomunikatow ,
								intTablicaKomunikatowZnacznikZapisu := intTablicaKomunikatowZnacznikZapisu ,
								intTablicaKomunikatowRozmiar := intTablicaKomunikatowRozmiar ,
								sWyslanyKomunikat := sWyslanyKomunikatDummy);
					sDane := '';
				END_IF	
			END_IF	
			IF fnKomunikatDaneSzukajWartosci(sKomunikat , 'VOLTL3=') = '?' OR fnKomunikatDaneSzukajWartosci(sKomunikat , 'ALL=') = '?' THEN
				fnKomunikatDaneDodaj_xOverFlow(sDane := sDane , sAtrybut := 'VOLTL3=' , sWartosc := REAL_TO_STRING(rNapiecieL3) , xOverFlow := xOverFlow);	
				IF xOverFlow = TRUE THEN
					fnZapiszKomunikat(	sCalyKomunikat := '' ,
								sTypKomunikatu := 'A' ,
								sMnemonik := sMnemonik ,
								sMACAdres := sMACAdres ,
								sIDNadawcy := sIdInstancji ,
								sIDOdbiorcy := sIdAplikacji ,
								sDaneZapasowe := sDaneZapasowe ,
								sDane := sDane ,
								arTablicaKomunikatow := arTablicaKomunikatow ,
								intTablicaKomunikatowZnacznikZapisu := intTablicaKomunikatowZnacznikZapisu ,
								intTablicaKomunikatowRozmiar := intTablicaKomunikatowRozmiar ,
								sWyslanyKomunikat := sWyslanyKomunikatDummy);
					sDane := '';
				END_IF	
			END_IF
			//Napięcia przewodowe
			IF fnKomunikatDaneSzukajWartosci(sKomunikat , 'VOLTL1L2=') = '?' OR fnKomunikatDaneSzukajWartosci(sKomunikat , 'ALL=') = '?' THEN
				fnKomunikatDaneDodaj_xOverFlow(sDane := sDane , sAtrybut := 'VOLTL1L2=' , sWartosc := REAL_TO_STRING(rNapiecieL1L2) , xOverFlow := xOverFlow);	
				IF xOverFlow = TRUE THEN
					fnZapiszKomunikat(	sCalyKomunikat := '' ,
								sTypKomunikatu := 'A' ,
								sMnemonik := sMnemonik ,
								sMACAdres := sMACAdres ,
								sIDNadawcy := sIdInstancji ,
								sIDOdbiorcy := sIdAplikacji ,
								sDaneZapasowe := sDaneZapasowe ,
								sDane := sDane ,
								arTablicaKomunikatow := arTablicaKomunikatow ,
								intTablicaKomunikatowZnacznikZapisu := intTablicaKomunikatowZnacznikZapisu ,
								intTablicaKomunikatowRozmiar := intTablicaKomunikatowRozmiar ,
								sWyslanyKomunikat := sWyslanyKomunikatDummy);
					sDane := '';
				END_IF	
			END_IF
			IF fnKomunikatDaneSzukajWartosci(sKomunikat , 'VOLTL2L3=') = '?' OR fnKomunikatDaneSzukajWartosci(sKomunikat , 'ALL=') = '?' THEN
				fnKomunikatDaneDodaj_xOverFlow(sDane := sDane , sAtrybut := 'VOLTL2L3=' , sWartosc := REAL_TO_STRING(rNapiecieL2L3) , xOverFlow := xOverFlow);	
				IF xOverFlow = TRUE THEN
					fnZapiszKomunikat(	sCalyKomunikat := '' ,
								sTypKomunikatu := 'A' ,
								sMnemonik := sMnemonik ,
								sMACAdres := sMACAdres ,
								sIDNadawcy := sIdInstancji ,
								sIDOdbiorcy := sIdAplikacji ,
								sDaneZapasowe := sDaneZapasowe ,
								sDane := sDane ,
								arTablicaKomunikatow := arTablicaKomunikatow ,
								intTablicaKomunikatowZnacznikZapisu := intTablicaKomunikatowZnacznikZapisu ,
								intTablicaKomunikatowRozmiar := intTablicaKomunikatowRozmiar ,
								sWyslanyKomunikat := sWyslanyKomunikatDummy);
					sDane := '';
				END_IF	
			END_IF	
			IF fnKomunikatDaneSzukajWartosci(sKomunikat , 'VOLTL3L1=') = '?' OR fnKomunikatDaneSzukajWartosci(sKomunikat , 'ALL=') = '?' THEN
				fnKomunikatDaneDodaj_xOverFlow(sDane := sDane , sAtrybut := 'VOLTL3L1=' , sWartosc := REAL_TO_STRING(rNapiecieL3L1) , xOverFlow := xOverFlow);	
				IF xOverFlow = TRUE THEN
					fnZapiszKomunikat(	sCalyKomunikat := '' ,
								sTypKomunikatu := 'A' ,
								sMnemonik := sMnemonik ,
								sMACAdres := sMACAdres ,
								sIDNadawcy := sIdInstancji ,
								sIDOdbiorcy := sIdAplikacji ,
								sDaneZapasowe := sDaneZapasowe ,
								sDane := sDane ,
								arTablicaKomunikatow := arTablicaKomunikatow ,
								intTablicaKomunikatowZnacznikZapisu := intTablicaKomunikatowZnacznikZapisu ,
								intTablicaKomunikatowRozmiar := intTablicaKomunikatowRozmiar ,
								sWyslanyKomunikat := sWyslanyKomunikatDummy);
					sDane := '';
				END_IF	
			END_IF
			//Częstotliwość 
			IF fnKomunikatDaneSzukajWartosci(sKomunikat , 'CZEST=') = '?' OR fnKomunikatDaneSzukajWartosci(sKomunikat , 'ALL=') = '?' THEN
				fnKomunikatDaneDodaj_xOverFlow(sDane := sDane , sAtrybut := 'CZEST=' , sWartosc := REAL_TO_STRING(rCzestotliwosc) , xOverFlow := xOverFlow);	
				IF xOverFlow = TRUE THEN
					fnZapiszKomunikat(	sCalyKomunikat := '' ,
								sTypKomunikatu := 'A' ,
								sMnemonik := sMnemonik ,
								sMACAdres := sMACAdres ,
								sIDNadawcy := sIdInstancji ,
								sIDOdbiorcy := sIdAplikacji ,
								sDaneZapasowe := sDaneZapasowe ,
								sDane := sDane ,
								arTablicaKomunikatow := arTablicaKomunikatow ,
								intTablicaKomunikatowZnacznikZapisu := intTablicaKomunikatowZnacznikZapisu ,
								intTablicaKomunikatowRozmiar := intTablicaKomunikatowRozmiar ,
								sWyslanyKomunikat := sWyslanyKomunikatDummy);
					sDane := '';
				END_IF	
			END_IF
			//Czas pracy 
			IF fnKomunikatDaneSzukajWartosci(sKomunikat , 'CZAS=') = '?' OR fnKomunikatDaneSzukajWartosci(sKomunikat , 'ALL=') = '?' THEN
				fnKomunikatDaneDodaj_xOverFlow(sDane := sDane , sAtrybut := 'CZAS=' , sWartosc := REAL_TO_STRING(rCzasPracyAnalizatora) , xOverFlow := xOverFlow);	
				IF xOverFlow = TRUE THEN
					fnZapiszKomunikat(	sCalyKomunikat := '' ,
								sTypKomunikatu := 'A' ,
								sMnemonik := sMnemonik ,
								sMACAdres := sMACAdres ,
								sIDNadawcy := sIdInstancji ,
								sIDOdbiorcy := sIdAplikacji ,
								sDaneZapasowe := sDaneZapasowe ,
								sDane := sDane ,
								arTablicaKomunikatow := arTablicaKomunikatow ,
								intTablicaKomunikatowZnacznikZapisu := intTablicaKomunikatowZnacznikZapisu ,
								intTablicaKomunikatowRozmiar := intTablicaKomunikatowRozmiar ,
								sWyslanyKomunikat := sWyslanyKomunikatDummy);
					sDane := '';
				END_IF	
			END_IF
			//Prądy fazowe
			IF fnKomunikatDaneSzukajWartosci(sKomunikat , 'AMPERL1=') = '?' OR fnKomunikatDaneSzukajWartosci(sKomunikat , 'ALL=') = '?' THEN
				fnKomunikatDaneDodaj_xOverFlow(sDane := sDane , sAtrybut := 'AMPERL1=' , sWartosc := REAL_TO_STRING(rPradL1) , xOverFlow := xOverFlow);	
				IF xOverFlow = TRUE THEN
					fnZapiszKomunikat(	sCalyKomunikat := '' ,
								sTypKomunikatu := 'A' ,
								sMnemonik := sMnemonik ,
								sMACAdres := sMACAdres ,
								sIDNadawcy := sIdInstancji ,
								sIDOdbiorcy := sIdAplikacji ,
								sDaneZapasowe := sDaneZapasowe ,
								sDane := sDane ,
								arTablicaKomunikatow := arTablicaKomunikatow ,
								intTablicaKomunikatowZnacznikZapisu := intTablicaKomunikatowZnacznikZapisu ,
								intTablicaKomunikatowRozmiar := intTablicaKomunikatowRozmiar ,
								sWyslanyKomunikat := sWyslanyKomunikatDummy);
					sDane := '';
				END_IF	
			END_IF
			IF fnKomunikatDaneSzukajWartosci(sKomunikat , 'AMPERL2=') = '?' OR fnKomunikatDaneSzukajWartosci(sKomunikat , 'ALL=') = '?' THEN
				fnKomunikatDaneDodaj_xOverFlow(sDane := sDane , sAtrybut := 'AMPERL2=' , sWartosc := REAL_TO_STRING(rPradL2) , xOverFlow := xOverFlow);	
				IF xOverFlow = TRUE THEN
					fnZapiszKomunikat(	sCalyKomunikat := '' ,
								sTypKomunikatu := 'A' ,
								sMnemonik := sMnemonik ,
								sMACAdres := sMACAdres ,
								sIDNadawcy := sIdInstancji ,
								sIDOdbiorcy := sIdAplikacji ,
								sDaneZapasowe := sDaneZapasowe ,
								sDane := sDane ,
								arTablicaKomunikatow := arTablicaKomunikatow ,
								intTablicaKomunikatowZnacznikZapisu := intTablicaKomunikatowZnacznikZapisu ,
								intTablicaKomunikatowRozmiar := intTablicaKomunikatowRozmiar ,
								sWyslanyKomunikat := sWyslanyKomunikatDummy);
					sDane := '';
				END_IF	
			END_IF	
			IF fnKomunikatDaneSzukajWartosci(sKomunikat , 'AMPERL3=') = '?' OR fnKomunikatDaneSzukajWartosci(sKomunikat , 'ALL=') = '?' THEN
				fnKomunikatDaneDodaj_xOverFlow(sDane := sDane , sAtrybut := 'AMPERL3=' , sWartosc := REAL_TO_STRING(rPradL3) , xOverFlow := xOverFlow);	
				IF xOverFlow = TRUE THEN
					fnZapiszKomunikat(	sCalyKomunikat := '' ,
								sTypKomunikatu := 'A' ,
								sMnemonik := sMnemonik ,
								sMACAdres := sMACAdres ,
								sIDNadawcy := sIdInstancji ,
								sIDOdbiorcy := sIdAplikacji ,
								sDaneZapasowe := sDaneZapasowe ,
								sDane := sDane ,
								arTablicaKomunikatow := arTablicaKomunikatow ,
								intTablicaKomunikatowZnacznikZapisu := intTablicaKomunikatowZnacznikZapisu ,
								intTablicaKomunikatowRozmiar := intTablicaKomunikatowRozmiar ,
								sWyslanyKomunikat := sWyslanyKomunikatDummy);
					sDane := '';
				END_IF	
			END_IF
			IF fnKomunikatDaneSzukajWartosci(sKomunikat , 'AMPERN=') = '?' OR fnKomunikatDaneSzukajWartosci(sKomunikat , 'ALL=') = '?' THEN
				fnKomunikatDaneDodaj_xOverFlow(sDane := sDane , sAtrybut := 'AMPERN=' , sWartosc := REAL_TO_STRING(rPradN) , xOverFlow := xOverFlow);	
				IF xOverFlow = TRUE THEN
					fnZapiszKomunikat(	sCalyKomunikat := '' ,
								sTypKomunikatu := 'A' ,
								sMnemonik := sMnemonik ,
								sMACAdres := sMACAdres ,
								sIDNadawcy := sIdInstancji ,
								sIDOdbiorcy := sIdAplikacji ,
								sDaneZapasowe := sDaneZapasowe ,
								sDane := sDane ,
								arTablicaKomunikatow := arTablicaKomunikatow ,
								intTablicaKomunikatowZnacznikZapisu := intTablicaKomunikatowZnacznikZapisu ,
								intTablicaKomunikatowRozmiar := intTablicaKomunikatowRozmiar ,
								sWyslanyKomunikat := sWyslanyKomunikatDummy);
					sDane := '';
				END_IF	
			END_IF
			//Prądy średnie fazowe
			IF fnKomunikatDaneSzukajWartosci(sKomunikat , 'AMPERAVGL1=') = '?' OR fnKomunikatDaneSzukajWartosci(sKomunikat , 'ALL=') = '?' THEN
				fnKomunikatDaneDodaj_xOverFlow(sDane := sDane , sAtrybut := 'AMPERAVGL1=' , sWartosc := REAL_TO_STRING(rPradSredniL1) , xOverFlow := xOverFlow);	
				IF xOverFlow = TRUE THEN
					fnZapiszKomunikat(	sCalyKomunikat := '' ,
								sTypKomunikatu := 'A' ,
								sMnemonik := sMnemonik ,
								sMACAdres := sMACAdres ,
								sIDNadawcy := sIdInstancji ,
								sIDOdbiorcy := sIdAplikacji ,
								sDaneZapasowe := sDaneZapasowe ,
								sDane := sDane ,
								arTablicaKomunikatow := arTablicaKomunikatow ,
								intTablicaKomunikatowZnacznikZapisu := intTablicaKomunikatowZnacznikZapisu ,
								intTablicaKomunikatowRozmiar := intTablicaKomunikatowRozmiar ,
								sWyslanyKomunikat := sWyslanyKomunikatDummy);
					sDane := '';
				END_IF	
			END_IF
			IF fnKomunikatDaneSzukajWartosci(sKomunikat , 'AMPERAVGL2=') = '?' OR fnKomunikatDaneSzukajWartosci(sKomunikat , 'ALL=') = '?' THEN
				fnKomunikatDaneDodaj_xOverFlow(sDane := sDane , sAtrybut := 'AMPERAVGL2=' , sWartosc := REAL_TO_STRING(rPradSredniL2) , xOverFlow := xOverFlow);	
				IF xOverFlow = TRUE THEN
					fnZapiszKomunikat(	sCalyKomunikat := '' ,
								sTypKomunikatu := 'A' ,
								sMnemonik := sMnemonik ,
								sMACAdres := sMACAdres ,
								sIDNadawcy := sIdInstancji ,
								sIDOdbiorcy := sIdAplikacji ,
								sDaneZapasowe := sDaneZapasowe ,
								sDane := sDane ,
								arTablicaKomunikatow := arTablicaKomunikatow ,
								intTablicaKomunikatowZnacznikZapisu := intTablicaKomunikatowZnacznikZapisu ,
								intTablicaKomunikatowRozmiar := intTablicaKomunikatowRozmiar ,
								sWyslanyKomunikat := sWyslanyKomunikatDummy);
					sDane := '';
				END_IF	
			END_IF	
			IF fnKomunikatDaneSzukajWartosci(sKomunikat , 'AMPERAVGL3=') = '?' OR fnKomunikatDaneSzukajWartosci(sKomunikat , 'ALL=') = '?' THEN
				fnKomunikatDaneDodaj_xOverFlow(sDane := sDane , sAtrybut := 'AMPERAVGL3=' , sWartosc := REAL_TO_STRING(rPradSredniL3) , xOverFlow := xOverFlow);	
				IF xOverFlow = TRUE THEN
					fnZapiszKomunikat(	sCalyKomunikat := '' ,
								sTypKomunikatu := 'A' ,
								sMnemonik := sMnemonik ,
								sMACAdres := sMACAdres ,
								sIDNadawcy := sIdInstancji ,
								sIDOdbiorcy := sIdAplikacji ,
								sDaneZapasowe := sDaneZapasowe ,
								sDane := sDane ,
								arTablicaKomunikatow := arTablicaKomunikatow ,
								intTablicaKomunikatowZnacznikZapisu := intTablicaKomunikatowZnacznikZapisu ,
								intTablicaKomunikatowRozmiar := intTablicaKomunikatowRozmiar ,
								sWyslanyKomunikat := sWyslanyKomunikatDummy);
					sDane := '';
				END_IF	
			END_IF
			//Prąd średni
			IF fnKomunikatDaneSzukajWartosci(sKomunikat , 'AMPERAVG=') = '?' OR fnKomunikatDaneSzukajWartosci(sKomunikat , 'ALL=') = '?' THEN
				fnKomunikatDaneDodaj_xOverFlow(sDane := sDane , sAtrybut := 'AMPERAVG=' , sWartosc := REAL_TO_STRING(rPradSredni) , xOverFlow := xOverFlow);	
				IF xOverFlow = TRUE THEN
					fnZapiszKomunikat(	sCalyKomunikat := '' ,
								sTypKomunikatu := 'A' ,
								sMnemonik := sMnemonik ,
								sMACAdres := sMACAdres ,
								sIDNadawcy := sIdInstancji ,
								sIDOdbiorcy := sIdAplikacji ,
								sDaneZapasowe := sDaneZapasowe ,
								sDane := sDane ,
								arTablicaKomunikatow := arTablicaKomunikatow ,
								intTablicaKomunikatowZnacznikZapisu := intTablicaKomunikatowZnacznikZapisu ,
								intTablicaKomunikatowRozmiar := intTablicaKomunikatowRozmiar ,
								sWyslanyKomunikat := sWyslanyKomunikatDummy);
					sDane := '';
				END_IF	
			END_IF
			//Moce 3-fazowe
			IF fnKomunikatDaneSzukajWartosci(sKomunikat , 'POWCE=') = '?' OR fnKomunikatDaneSzukajWartosci(sKomunikat , 'ALL=') = '?' THEN
				fnKomunikatDaneDodaj_xOverFlow(sDane := sDane , sAtrybut := '=' , sWartosc := REAL_TO_STRING(rMocCzynnaCalkowita) , xOverFlow := xOverFlow);	
				IF xOverFlow = TRUE THEN
					fnZapiszKomunikat(	sCalyKomunikat := '' ,
								sTypKomunikatu := 'A' ,
								sMnemonik := sMnemonik ,
								sMACAdres := sMACAdres ,
								sIDNadawcy := sIdInstancji ,
								sIDOdbiorcy := sIdAplikacji ,
								sDaneZapasowe := sDaneZapasowe ,
								sDane := sDane ,
								arTablicaKomunikatow := arTablicaKomunikatow ,
								intTablicaKomunikatowZnacznikZapisu := intTablicaKomunikatowZnacznikZapisu ,
								intTablicaKomunikatowRozmiar := intTablicaKomunikatowRozmiar ,
								sWyslanyKomunikat := sWyslanyKomunikatDummy);
					sDane := '';
				END_IF	
			END_IF
			IF fnKomunikatDaneSzukajWartosci(sKomunikat , 'POWBE=') = '?' OR fnKomunikatDaneSzukajWartosci(sKomunikat , 'ALL=') = '?' THEN
				fnKomunikatDaneDodaj_xOverFlow(sDane := sDane , sAtrybut := 'POWBE=' , sWartosc := REAL_TO_STRING(rMocBiernaCalkowita) , xOverFlow := xOverFlow);	
				IF xOverFlow = TRUE THEN
					fnZapiszKomunikat(	sCalyKomunikat := '' ,
								sTypKomunikatu := 'A' ,
								sMnemonik := sMnemonik ,
								sMACAdres := sMACAdres ,
								sIDNadawcy := sIdInstancji ,
								sIDOdbiorcy := sIdAplikacji ,
								sDaneZapasowe := sDaneZapasowe ,
								sDane := sDane ,
								arTablicaKomunikatow := arTablicaKomunikatow ,
								intTablicaKomunikatowZnacznikZapisu := intTablicaKomunikatowZnacznikZapisu ,
								intTablicaKomunikatowRozmiar := intTablicaKomunikatowRozmiar ,
								sWyslanyKomunikat := sWyslanyKomunikatDummy);
					sDane := '';
				END_IF	
			END_IF	
			IF fnKomunikatDaneSzukajWartosci(sKomunikat , 'POWPE=') = '?' OR fnKomunikatDaneSzukajWartosci(sKomunikat , 'ALL=') = '?' THEN
				fnKomunikatDaneDodaj_xOverFlow(sDane := sDane , sAtrybut := 'POWPE=' , sWartosc := REAL_TO_STRING(rMocPozornaCalkowita) , xOverFlow := xOverFlow);	
				IF xOverFlow = TRUE THEN
					fnZapiszKomunikat(	sCalyKomunikat := '' ,
								sTypKomunikatu := 'A' ,
								sMnemonik := sMnemonik ,
								sMACAdres := sMACAdres ,
								sIDNadawcy := sIdInstancji ,
								sIDOdbiorcy := sIdAplikacji ,
								sDaneZapasowe := sDaneZapasowe ,
								sDane := sDane ,
								arTablicaKomunikatow := arTablicaKomunikatow ,
								intTablicaKomunikatowZnacznikZapisu := intTablicaKomunikatowZnacznikZapisu ,
								intTablicaKomunikatowRozmiar := intTablicaKomunikatowRozmiar ,
								sWyslanyKomunikat := sWyslanyKomunikatDummy);
					sDane := '';
				END_IF	
			END_IF
			//Współczynnik mocy 3-fazowy
			IF fnKomunikatDaneSzukajWartosci(sKomunikat , 'FACTOR3PH=') = '?' OR fnKomunikatDaneSzukajWartosci(sKomunikat , 'ALL=') = '?' THEN
				fnKomunikatDaneDodaj_xOverFlow(sDane := sDane , sAtrybut := 'FACTOR3PH=' , sWartosc := REAL_TO_STRING(rWspolczynnikMocyCalkowity) , xOverFlow := xOverFlow);
				IF xOverFlow = TRUE THEN
					fnZapiszKomunikat(	sCalyKomunikat := '' ,
								sTypKomunikatu := 'A' ,
								sMnemonik := sMnemonik ,
								sMACAdres := sMACAdres ,
								sIDNadawcy := sIdInstancji ,
								sIDOdbiorcy := sIdAplikacji ,
								sDaneZapasowe := sDaneZapasowe ,
								sDane := sDane ,
								arTablicaKomunikatow := arTablicaKomunikatow ,
								intTablicaKomunikatowZnacznikZapisu := intTablicaKomunikatowZnacznikZapisu ,
								intTablicaKomunikatowRozmiar := intTablicaKomunikatowRozmiar ,
								sWyslanyKomunikat := sWyslanyKomunikatDummy);
					sDane := '';
				END_IF		
			END_IF
			//Moce czynne fazowe
			IF fnKomunikatDaneSzukajWartosci(sKomunikat , 'POWCECL1=') = '?' OR fnKomunikatDaneSzukajWartosci(sKomunikat , 'ALL=') = '?' THEN
				fnKomunikatDaneDodaj_xOverFlow(sDane := sDane , sAtrybut := 'CL1=' , sWartosc := REAL_TO_STRING(rMocCzynnaL1) , xOverFlow := xOverFlow);	
				IF xOverFlow = TRUE THEN
					fnZapiszKomunikat(	sCalyKomunikat := '' ,
								sTypKomunikatu := 'A' ,
								sMnemonik := sMnemonik ,
								sMACAdres := sMACAdres ,
								sIDNadawcy := sIdInstancji ,
								sIDOdbiorcy := sIdAplikacji ,
								sDaneZapasowe := sDaneZapasowe ,
								sDane := sDane ,
								arTablicaKomunikatow := arTablicaKomunikatow ,
								intTablicaKomunikatowZnacznikZapisu := intTablicaKomunikatowZnacznikZapisu ,
								intTablicaKomunikatowRozmiar := intTablicaKomunikatowRozmiar ,
								sWyslanyKomunikat := sWyslanyKomunikatDummy);
					sDane := '';
				END_IF	
			END_IF
			IF fnKomunikatDaneSzukajWartosci(sKomunikat , 'POWCECL2=') = '?' OR fnKomunikatDaneSzukajWartosci(sKomunikat , 'ALL=') = '?' THEN
				fnKomunikatDaneDodaj_xOverFlow(sDane := sDane , sAtrybut := 'CL2=' , sWartosc := REAL_TO_STRING(rMocCzynnaL2) , xOverFlow := xOverFlow);	
				IF xOverFlow = TRUE THEN
					fnZapiszKomunikat(	sCalyKomunikat := '' ,
								sTypKomunikatu := 'A' ,
								sMnemonik := sMnemonik ,
								sMACAdres := sMACAdres ,
								sIDNadawcy := sIdInstancji ,
								sIDOdbiorcy := sIdAplikacji ,
								sDaneZapasowe := sDaneZapasowe ,
								sDane := sDane ,
								arTablicaKomunikatow := arTablicaKomunikatow ,
								intTablicaKomunikatowZnacznikZapisu := intTablicaKomunikatowZnacznikZapisu ,
								intTablicaKomunikatowRozmiar := intTablicaKomunikatowRozmiar ,
								sWyslanyKomunikat := sWyslanyKomunikatDummy);
					sDane := '';
				END_IF	
			END_IF	
			IF fnKomunikatDaneSzukajWartosci(sKomunikat , 'POWCECL3=') = '?' OR fnKomunikatDaneSzukajWartosci(sKomunikat , 'ALL=') = '?' THEN
				fnKomunikatDaneDodaj_xOverFlow(sDane := sDane , sAtrybut := 'CL3=' , sWartosc := REAL_TO_STRING(rMocCzynnaL3) , xOverFlow := xOverFlow);
				IF xOverFlow = TRUE THEN
					fnZapiszKomunikat(	sCalyKomunikat := '' ,
								sTypKomunikatu := 'A' ,
								sMnemonik := sMnemonik ,
								sMACAdres := sMACAdres ,
								sIDNadawcy := sIdInstancji ,
								sIDOdbiorcy := sIdAplikacji ,
								sDaneZapasowe := sDaneZapasowe ,
								sDane := sDane ,
								arTablicaKomunikatow := arTablicaKomunikatow ,
								intTablicaKomunikatowZnacznikZapisu := intTablicaKomunikatowZnacznikZapisu ,
								intTablicaKomunikatowRozmiar := intTablicaKomunikatowRozmiar ,
								sWyslanyKomunikat := sWyslanyKomunikatDummy);
					sDane := '';
				END_IF		
			END_IF
			//Moce bierne fazowe
			IF fnKomunikatDaneSzukajWartosci(sKomunikat , 'POWCEBL1=') = '?' OR fnKomunikatDaneSzukajWartosci(sKomunikat , 'ALL=') = '?' THEN
				fnKomunikatDaneDodaj_xOverFlow(sDane := sDane , sAtrybut := 'BL1=' , sWartosc := REAL_TO_STRING(rMocBiernaL1) , xOverFlow := xOverFlow);	
				IF xOverFlow = TRUE THEN
					fnZapiszKomunikat(	sCalyKomunikat := '' ,
								sTypKomunikatu := 'A' ,
								sMnemonik := sMnemonik ,
								sMACAdres := sMACAdres ,
								sIDNadawcy := sIdInstancji ,
								sIDOdbiorcy := sIdAplikacji ,
								sDaneZapasowe := sDaneZapasowe ,
								sDane := sDane ,
								arTablicaKomunikatow := arTablicaKomunikatow ,
								intTablicaKomunikatowZnacznikZapisu := intTablicaKomunikatowZnacznikZapisu ,
								intTablicaKomunikatowRozmiar := intTablicaKomunikatowRozmiar ,
								sWyslanyKomunikat := sWyslanyKomunikatDummy);
					sDane := '';
				END_IF	
			END_IF
			IF fnKomunikatDaneSzukajWartosci(sKomunikat , 'POWCEBL2=') = '?' OR fnKomunikatDaneSzukajWartosci(sKomunikat , 'ALL=') = '?' THEN
				fnKomunikatDaneDodaj_xOverFlow(sDane := sDane , sAtrybut := 'POWCEBL2=' , sWartosc := REAL_TO_STRING(rMocBiernaL2) , xOverFlow := xOverFlow);	
				IF xOverFlow = TRUE THEN
					fnZapiszKomunikat(	sCalyKomunikat := '' ,
								sTypKomunikatu := 'A' ,
								sMnemonik := sMnemonik ,
								sMACAdres := sMACAdres ,
								sIDNadawcy := sIdInstancji ,
								sIDOdbiorcy := sIdAplikacji ,
								sDaneZapasowe := sDaneZapasowe ,
								sDane := sDane ,
								arTablicaKomunikatow := arTablicaKomunikatow ,
								intTablicaKomunikatowZnacznikZapisu := intTablicaKomunikatowZnacznikZapisu ,
								intTablicaKomunikatowRozmiar := intTablicaKomunikatowRozmiar ,
								sWyslanyKomunikat := sWyslanyKomunikatDummy);
					sDane := '';
				END_IF	
			END_IF	
			IF fnKomunikatDaneSzukajWartosci(sKomunikat , 'POWCEBL3=') = '?' OR fnKomunikatDaneSzukajWartosci(sKomunikat , 'ALL=') = '?' THEN
				fnKomunikatDaneDodaj_xOverFlow(sDane := sDane , sAtrybut := 'POWCEBL3=' , sWartosc := REAL_TO_STRING(rMocBiernaL3) , xOverFlow := xOverFlow);	
				IF xOverFlow = TRUE THEN
					fnZapiszKomunikat(	sCalyKomunikat := '' ,
								sTypKomunikatu := 'A' ,
								sMnemonik := sMnemonik ,
								sMACAdres := sMACAdres ,
								sIDNadawcy := sIdInstancji ,
								sIDOdbiorcy := sIdAplikacji ,
								sDaneZapasowe := sDaneZapasowe ,
								sDane := sDane ,
								arTablicaKomunikatow := arTablicaKomunikatow ,
								intTablicaKomunikatowZnacznikZapisu := intTablicaKomunikatowZnacznikZapisu ,
								intTablicaKomunikatowRozmiar := intTablicaKomunikatowRozmiar ,
								sWyslanyKomunikat := sWyslanyKomunikatDummy);
					sDane := '';
				END_IF	
			END_IF
			//Moce pozorne fazowe
			IF fnKomunikatDaneSzukajWartosci(sKomunikat , 'POWCEPL1=') = '?' OR fnKomunikatDaneSzukajWartosci(sKomunikat , 'ALL=') = '?' THEN
				fnKomunikatDaneDodaj_xOverFlow(sDane := sDane , sAtrybut := 'POWCEPL1=' , sWartosc := REAL_TO_STRING(rMocPozornaL1) , xOverFlow := xOverFlow);	
				IF xOverFlow = TRUE THEN
					fnZapiszKomunikat(	sCalyKomunikat := '' ,
								sTypKomunikatu := 'A' ,
								sMnemonik := sMnemonik ,
								sMACAdres := sMACAdres ,
								sIDNadawcy := sIdInstancji ,
								sIDOdbiorcy := sIdAplikacji ,
								sDaneZapasowe := sDaneZapasowe ,
								sDane := sDane ,
								arTablicaKomunikatow := arTablicaKomunikatow ,
								intTablicaKomunikatowZnacznikZapisu := intTablicaKomunikatowZnacznikZapisu ,
								intTablicaKomunikatowRozmiar := intTablicaKomunikatowRozmiar ,
								sWyslanyKomunikat := sWyslanyKomunikatDummy);
					sDane := '';
				END_IF	
			END_IF
			IF fnKomunikatDaneSzukajWartosci(sKomunikat , 'POWCEPL2=') = '?' OR fnKomunikatDaneSzukajWartosci(sKomunikat , 'ALL=') = '?' THEN
				fnKomunikatDaneDodaj_xOverFlow(sDane := sDane , sAtrybut := 'POWCEPL2=' , sWartosc := REAL_TO_STRING(rMocPozornaL2) , xOverFlow := xOverFlow);	
				IF xOverFlow = TRUE THEN
					fnZapiszKomunikat(	sCalyKomunikat := '' ,
								sTypKomunikatu := 'A' ,
								sMnemonik := sMnemonik ,
								sMACAdres := sMACAdres ,
								sIDNadawcy := sIdInstancji ,
								sIDOdbiorcy := sIdAplikacji ,
								sDaneZapasowe := sDaneZapasowe ,
								sDane := sDane ,
								arTablicaKomunikatow := arTablicaKomunikatow ,
								intTablicaKomunikatowZnacznikZapisu := intTablicaKomunikatowZnacznikZapisu ,
								intTablicaKomunikatowRozmiar := intTablicaKomunikatowRozmiar ,
								sWyslanyKomunikat := sWyslanyKomunikatDummy);
					sDane := '';
				END_IF	
			END_IF	
			IF fnKomunikatDaneSzukajWartosci(sKomunikat , 'POWCEPL3=') = '?' OR fnKomunikatDaneSzukajWartosci(sKomunikat , 'ALL=') = '?' THEN
				fnKomunikatDaneDodaj_xOverFlow(sDane := sDane , sAtrybut := 'POWCEPL3=' , sWartosc := REAL_TO_STRING(rMocPozornaL3) , xOverFlow := xOverFlow);	
				IF xOverFlow = TRUE THEN
					fnZapiszKomunikat(	sCalyKomunikat := '' ,
								sTypKomunikatu := 'A' ,
								sMnemonik := sMnemonik ,
								sMACAdres := sMACAdres ,
								sIDNadawcy := sIdInstancji ,
								sIDOdbiorcy := sIdAplikacji ,
								sDaneZapasowe := sDaneZapasowe ,
								sDane := sDane ,
								arTablicaKomunikatow := arTablicaKomunikatow ,
								intTablicaKomunikatowZnacznikZapisu := intTablicaKomunikatowZnacznikZapisu ,
								intTablicaKomunikatowRozmiar := intTablicaKomunikatowRozmiar ,
								sWyslanyKomunikat := sWyslanyKomunikatDummy);
					sDane := '';
				END_IF	
			END_IF
			//Współczynniki mocy fazowe
			IF fnKomunikatDaneSzukajWartosci(sKomunikat , 'FACTORL1=') = '?' OR fnKomunikatDaneSzukajWartosci(sKomunikat , 'ALL=') = '?' THEN
				fnKomunikatDaneDodaj_xOverFlow(sDane := sDane , sAtrybut := 'FACTORL1=' , sWartosc := REAL_TO_STRING(rWspolczynnikMocyL1) , xOverFlow := xOverFlow);	
				IF xOverFlow = TRUE THEN
					fnZapiszKomunikat(	sCalyKomunikat := '' ,
								sTypKomunikatu := 'A' ,
								sMnemonik := sMnemonik ,
								sMACAdres := sMACAdres ,
								sIDNadawcy := sIdInstancji ,
								sIDOdbiorcy := sIdAplikacji ,
								sDaneZapasowe := sDaneZapasowe ,
								sDane := sDane ,
								arTablicaKomunikatow := arTablicaKomunikatow ,
								intTablicaKomunikatowZnacznikZapisu := intTablicaKomunikatowZnacznikZapisu ,
								intTablicaKomunikatowRozmiar := intTablicaKomunikatowRozmiar ,
								sWyslanyKomunikat := sWyslanyKomunikatDummy);
					sDane := '';
				END_IF	
			END_IF
			IF fnKomunikatDaneSzukajWartosci(sKomunikat , 'FACTORL2=') = '?' OR fnKomunikatDaneSzukajWartosci(sKomunikat , 'ALL=') = '?' THEN
				fnKomunikatDaneDodaj_xOverFlow(sDane := sDane , sAtrybut := 'FACTORL2=' , sWartosc := REAL_TO_STRING(rWspolczynnikMocyL2) , xOverFlow := xOverFlow);
				IF xOverFlow = TRUE THEN
					fnZapiszKomunikat(	sCalyKomunikat := '' ,
								sTypKomunikatu := 'A' ,
								sMnemonik := sMnemonik ,
								sMACAdres := sMACAdres ,
								sIDNadawcy := sIdInstancji ,
								sIDOdbiorcy := sIdAplikacji ,
								sDaneZapasowe := sDaneZapasowe ,
								sDane := sDane ,
								arTablicaKomunikatow := arTablicaKomunikatow ,
								intTablicaKomunikatowZnacznikZapisu := intTablicaKomunikatowZnacznikZapisu ,
								intTablicaKomunikatowRozmiar := intTablicaKomunikatowRozmiar ,
								sWyslanyKomunikat := sWyslanyKomunikatDummy);
					sDane := '';
				END_IF		
			END_IF
			IF fnKomunikatDaneSzukajWartosci(sKomunikat , 'FACTORL3=') = '?' OR fnKomunikatDaneSzukajWartosci(sKomunikat , 'ALL=') = '?' THEN
				fnKomunikatDaneDodaj_xOverFlow(sDane := sDane , sAtrybut := 'FACTORL3=' , sWartosc := REAL_TO_STRING(rWspolczynnikMocyL3) , xOverFlow := xOverFlow);	
				IF xOverFlow = TRUE THEN
					fnZapiszKomunikat(	sCalyKomunikat := '' ,
								sTypKomunikatu := 'A' ,
								sMnemonik := sMnemonik ,
								sMACAdres := sMACAdres ,
								sIDNadawcy := sIdInstancji ,
								sIDOdbiorcy := sIdAplikacji ,
								sDaneZapasowe := sDaneZapasowe ,
								sDane := sDane ,
								arTablicaKomunikatow := arTablicaKomunikatow ,
								intTablicaKomunikatowZnacznikZapisu := intTablicaKomunikatowZnacznikZapisu ,
								intTablicaKomunikatowRozmiar := intTablicaKomunikatowRozmiar ,
								sWyslanyKomunikat := sWyslanyKomunikatDummy);
					sDane := '';
				END_IF	
			END_IF
			//Energia pobrana
			IF fnKomunikatDaneSzukajWartosci(sKomunikat , 'ENCE=') = '?' OR fnKomunikatDaneSzukajWartosci(sKomunikat , 'ALL=') = '?' THEN
				fnKomunikatDaneDodaj_xOverFlow(sDane := sDane , sAtrybut := 'ENCE=' , sWartosc := REAL_TO_STRING(rEnergiaCzynnaPobrana) , xOverFlow := xOverFlow);	
				IF xOverFlow = TRUE THEN
					fnZapiszKomunikat(	sCalyKomunikat := '' ,
								sTypKomunikatu := 'A' ,
								sMnemonik := sMnemonik ,
								sMACAdres := sMACAdres ,
								sIDNadawcy := sIdInstancji ,
								sIDOdbiorcy := sIdAplikacji ,
								sDaneZapasowe := sDaneZapasowe ,
								sDane := sDane ,
								arTablicaKomunikatow := arTablicaKomunikatow ,
								intTablicaKomunikatowZnacznikZapisu := intTablicaKomunikatowZnacznikZapisu ,
								intTablicaKomunikatowRozmiar := intTablicaKomunikatowRozmiar ,
								sWyslanyKomunikat := sWyslanyKomunikatDummy);
					sDane := '';
				END_IF	
			END_IF
			IF fnKomunikatDaneSzukajWartosci(sKomunikat , 'ENBE=') = '?' OR fnKomunikatDaneSzukajWartosci(sKomunikat , 'ALL=') = '?' THEN
				fnKomunikatDaneDodaj_xOverFlow(sDane := sDane , sAtrybut := 'ENBE=' , sWartosc := REAL_TO_STRING(rEnergiaBiernaPobrana) , xOverFlow := xOverFlow);	
				IF xOverFlow = TRUE THEN
					fnZapiszKomunikat(	sCalyKomunikat := '' ,
								sTypKomunikatu := 'A' ,
								sMnemonik := sMnemonik ,
								sMACAdres := sMACAdres ,
								sIDNadawcy := sIdInstancji ,
								sIDOdbiorcy := sIdAplikacji ,
								sDaneZapasowe := sDaneZapasowe ,
								sDane := sDane ,
								arTablicaKomunikatow := arTablicaKomunikatow ,
								intTablicaKomunikatowZnacznikZapisu := intTablicaKomunikatowZnacznikZapisu ,
								intTablicaKomunikatowRozmiar := intTablicaKomunikatowRozmiar ,
								sWyslanyKomunikat := sWyslanyKomunikatDummy);
					sDane := '';
				END_IF	
			END_IF
			IF fnKomunikatDaneSzukajWartosci(sKomunikat , 'ENPE=') = '?' OR fnKomunikatDaneSzukajWartosci(sKomunikat , 'ALL=') = '?' THEN
				fnKomunikatDaneDodaj_xOverFlow(sDane := sDane , sAtrybut := 'ENPE=' , sWartosc := REAL_TO_STRING(rEnergiaPozornaPobrana) , xOverFlow := xOverFlow);	
				IF xOverFlow = TRUE THEN
					fnZapiszKomunikat(	sCalyKomunikat := '' ,
								sTypKomunikatu := 'A' ,
								sMnemonik := sMnemonik ,
								sMACAdres := sMACAdres ,
								sIDNadawcy := sIdInstancji ,
								sIDOdbiorcy := sIdAplikacji ,
								sDaneZapasowe := sDaneZapasowe ,
								sDane := sDane ,
								arTablicaKomunikatow := arTablicaKomunikatow ,
								intTablicaKomunikatowZnacznikZapisu := intTablicaKomunikatowZnacznikZapisu ,
								intTablicaKomunikatowRozmiar := intTablicaKomunikatowRozmiar ,
								sWyslanyKomunikat := sWyslanyKomunikatDummy);
					sDane := '';
				END_IF	
			END_IF
			//Moce średnie
			IF fnKomunikatDaneSzukajWartosci(sKomunikat , 'POWAVGEC=') = '?' OR fnKomunikatDaneSzukajWartosci(sKomunikat , 'ALL=') = '?' THEN
				fnKomunikatDaneDodaj_xOverFlow(sDane := sDane , sAtrybut := 'POWAVGEC=' , sWartosc := REAL_TO_STRING(rMocCzynnaSrednia) , xOverFlow := xOverFlow);	
				IF xOverFlow = TRUE THEN
					fnZapiszKomunikat(	sCalyKomunikat := '' ,
								sTypKomunikatu := 'A' ,
								sMnemonik := sMnemonik ,
								sMACAdres := sMACAdres ,
								sIDNadawcy := sIdInstancji ,
								sIDOdbiorcy := sIdAplikacji ,
								sDaneZapasowe := sDaneZapasowe ,
								sDane := sDane ,
								arTablicaKomunikatow := arTablicaKomunikatow ,
								intTablicaKomunikatowZnacznikZapisu := intTablicaKomunikatowZnacznikZapisu ,
								intTablicaKomunikatowRozmiar := intTablicaKomunikatowRozmiar ,
								sWyslanyKomunikat := sWyslanyKomunikatDummy);
					sDane := '';
				END_IF	
			END_IF
			IF fnKomunikatDaneSzukajWartosci(sKomunikat , 'POWAVGEB=') = '?' OR fnKomunikatDaneSzukajWartosci(sKomunikat , 'ALL=') = '?' THEN
				fnKomunikatDaneDodaj_xOverFlow(sDane := sDane , sAtrybut := 'POWAVGEB=' , sWartosc := REAL_TO_STRING(rMocBiernaSrednia) , xOverFlow := xOverFlow);	
				IF xOverFlow = TRUE THEN
					fnZapiszKomunikat(	sCalyKomunikat := '' ,
								sTypKomunikatu := 'A' ,
								sMnemonik := sMnemonik ,
								sMACAdres := sMACAdres ,
								sIDNadawcy := sIdInstancji ,
								sIDOdbiorcy := sIdAplikacji ,
								sDaneZapasowe := sDaneZapasowe ,
								sDane := sDane ,
								arTablicaKomunikatow := arTablicaKomunikatow ,
								intTablicaKomunikatowZnacznikZapisu := intTablicaKomunikatowZnacznikZapisu ,
								intTablicaKomunikatowRozmiar := intTablicaKomunikatowRozmiar ,
								sWyslanyKomunikat := sWyslanyKomunikatDummy);
					sDane := '';
				END_IF	
			END_IF	
			IF fnKomunikatDaneSzukajWartosci(sKomunikat , 'POWAVGEP=') = '?' OR fnKomunikatDaneSzukajWartosci(sKomunikat , 'ALL=') = '?' THEN
				fnKomunikatDaneDodaj_xOverFlow(sDane := sDane , sAtrybut := 'POWAVGCEP=' , sWartosc := REAL_TO_STRING(rMocPozornaSrednia) , xOverFlow := xOverFlow);	
				IF xOverFlow = TRUE THEN
					fnZapiszKomunikat(	sCalyKomunikat := '' ,
								sTypKomunikatu := 'A' ,
								sMnemonik := sMnemonik ,
								sMACAdres := sMACAdres ,
								sIDNadawcy := sIdInstancji ,
								sIDOdbiorcy := sIdAplikacji ,
								sDaneZapasowe := sDaneZapasowe ,
								sDane := sDane ,
								arTablicaKomunikatow := arTablicaKomunikatow ,
								intTablicaKomunikatowZnacznikZapisu := intTablicaKomunikatowZnacznikZapisu ,
								intTablicaKomunikatowRozmiar := intTablicaKomunikatowRozmiar ,
								sWyslanyKomunikat := sWyslanyKomunikatDummy);
					sDane := '';
				END_IF	
			END_IF
			//Napięcia maksymalne fazowe
			IF fnKomunikatDaneSzukajWartosci(sKomunikat , 'VOLTMAXL1=') = '?' OR fnKomunikatDaneSzukajWartosci(sKomunikat , 'ALL=') = '?' THEN
				fnKomunikatDaneDodaj_xOverFlow(sDane := sDane , sAtrybut := 'VOLTMAXL1=' , sWartosc := REAL_TO_STRING(rMaksymalneNapiecieL1) , xOverFlow := xOverFlow);	
				IF xOverFlow = TRUE THEN
					fnZapiszKomunikat(	sCalyKomunikat := '' ,
								sTypKomunikatu := 'A' ,
								sMnemonik := sMnemonik ,
								sMACAdres := sMACAdres ,
								sIDNadawcy := sIdInstancji ,
								sIDOdbiorcy := sIdAplikacji ,
								sDaneZapasowe := sDaneZapasowe ,
								sDane := sDane ,
								arTablicaKomunikatow := arTablicaKomunikatow ,
								intTablicaKomunikatowZnacznikZapisu := intTablicaKomunikatowZnacznikZapisu ,
								intTablicaKomunikatowRozmiar := intTablicaKomunikatowRozmiar ,
								sWyslanyKomunikat := sWyslanyKomunikatDummy);
					sDane := '';
				END_IF	
			END_IF
			IF fnKomunikatDaneSzukajWartosci(sKomunikat , 'VOLTMAXL2=') = '?' OR fnKomunikatDaneSzukajWartosci(sKomunikat , 'ALL=') = '?' THEN
				fnKomunikatDaneDodaj_xOverFlow(sDane := sDane , sAtrybut := 'VOLTMAXL2=' , sWartosc := REAL_TO_STRING(rMaksymalneNapiecieL2) , xOverFlow := xOverFlow);	
				IF xOverFlow = TRUE THEN
					fnZapiszKomunikat(	sCalyKomunikat := '' ,
								sTypKomunikatu := 'A' ,
								sMnemonik := sMnemonik ,
								sMACAdres := sMACAdres ,
								sIDNadawcy := sIdInstancji ,
								sIDOdbiorcy := sIdAplikacji ,
								sDaneZapasowe := sDaneZapasowe ,
								sDane := sDane ,
								arTablicaKomunikatow := arTablicaKomunikatow ,
								intTablicaKomunikatowZnacznikZapisu := intTablicaKomunikatowZnacznikZapisu ,
								intTablicaKomunikatowRozmiar := intTablicaKomunikatowRozmiar ,
								sWyslanyKomunikat := sWyslanyKomunikatDummy);
					sDane := '';
				END_IF	
			END_IF	
			IF fnKomunikatDaneSzukajWartosci(sKomunikat , 'VOLTMAXL3=') = '?' OR fnKomunikatDaneSzukajWartosci(sKomunikat , 'ALL=') = '?' THEN
				fnKomunikatDaneDodaj_xOverFlow(sDane := sDane , sAtrybut := 'VOLTMAXL3=' , sWartosc := REAL_TO_STRING(rMaksymalneNapiecieL3) , xOverFlow := xOverFlow);	
				IF xOverFlow = TRUE THEN
					fnZapiszKomunikat(	sCalyKomunikat := '' ,
								sTypKomunikatu := 'A' ,
								sMnemonik := sMnemonik ,
								sMACAdres := sMACAdres ,
								sIDNadawcy := sIdInstancji ,
								sIDOdbiorcy := sIdAplikacji ,
								sDaneZapasowe := sDaneZapasowe ,
								sDane := sDane ,
								arTablicaKomunikatow := arTablicaKomunikatow ,
								intTablicaKomunikatowZnacznikZapisu := intTablicaKomunikatowZnacznikZapisu ,
								intTablicaKomunikatowRozmiar := intTablicaKomunikatowRozmiar ,
								sWyslanyKomunikat := sWyslanyKomunikatDummy);
					sDane := '';
				END_IF	
			END_IF
			//THD napięcia, fazowe
			IF fnKomunikatDaneSzukajWartosci(sKomunikat , 'VOLTTHDL1=') = '?' OR fnKomunikatDaneSzukajWartosci(sKomunikat , 'ALL=') = '?' THEN
				fnKomunikatDaneDodaj_xOverFlow(sDane := sDane , sAtrybut := 'VOLTTHDL1=' , sWartosc := REAL_TO_STRING(rTHDNapieciaL1) , xOverFlow := xOverFlow);	
				IF xOverFlow = TRUE THEN
					fnZapiszKomunikat(	sCalyKomunikat := '' ,
								sTypKomunikatu := 'A' ,
								sMnemonik := sMnemonik ,
								sMACAdres := sMACAdres ,
								sIDNadawcy := sIdInstancji ,
								sIDOdbiorcy := sIdAplikacji ,
								sDaneZapasowe := sDaneZapasowe ,
								sDane := sDane ,
								arTablicaKomunikatow := arTablicaKomunikatow ,
								intTablicaKomunikatowZnacznikZapisu := intTablicaKomunikatowZnacznikZapisu ,
								intTablicaKomunikatowRozmiar := intTablicaKomunikatowRozmiar ,
								sWyslanyKomunikat := sWyslanyKomunikatDummy);
					sDane := '';
				END_IF	
			END_IF
			IF fnKomunikatDaneSzukajWartosci(sKomunikat , 'VOLTTHDL2=') = '?' OR fnKomunikatDaneSzukajWartosci(sKomunikat , 'ALL=') = '?' THEN
				fnKomunikatDaneDodaj_xOverFlow(sDane := sDane , sAtrybut := 'VOLTTHDL2=' , sWartosc := REAL_TO_STRING(rTHDNapieciaL2) , xOverFlow := xOverFlow);	
				IF xOverFlow = TRUE THEN
					fnZapiszKomunikat(	sCalyKomunikat := '' ,
								sTypKomunikatu := 'A' ,
								sMnemonik := sMnemonik ,
								sMACAdres := sMACAdres ,
								sIDNadawcy := sIdInstancji ,
								sIDOdbiorcy := sIdAplikacji ,
								sDaneZapasowe := sDaneZapasowe ,
								sDane := sDane ,
								arTablicaKomunikatow := arTablicaKomunikatow ,
								intTablicaKomunikatowZnacznikZapisu := intTablicaKomunikatowZnacznikZapisu ,
								intTablicaKomunikatowRozmiar := intTablicaKomunikatowRozmiar ,
								sWyslanyKomunikat := sWyslanyKomunikatDummy);
					sDane := '';
				END_IF	
			END_IF	
			IF fnKomunikatDaneSzukajWartosci(sKomunikat , 'VOLTTHDL3=') = '?' OR fnKomunikatDaneSzukajWartosci(sKomunikat , 'ALL=') = '?' THEN
				fnKomunikatDaneDodaj_xOverFlow(sDane := sDane , sAtrybut := 'VOLTTHDL3=' , sWartosc := REAL_TO_STRING(rTHDNapieciaL3) , xOverFlow := xOverFlow);
				IF xOverFlow = TRUE THEN
					fnZapiszKomunikat(	sCalyKomunikat := '' ,
								sTypKomunikatu := 'A' ,
								sMnemonik := sMnemonik ,
								sMACAdres := sMACAdres ,
								sIDNadawcy := sIdInstancji ,
								sIDOdbiorcy := sIdAplikacji ,
								sDaneZapasowe := sDaneZapasowe ,
								sDane := sDane ,
								arTablicaKomunikatow := arTablicaKomunikatow ,
								intTablicaKomunikatowZnacznikZapisu := intTablicaKomunikatowZnacznikZapisu ,
								intTablicaKomunikatowRozmiar := intTablicaKomunikatowRozmiar ,
								sWyslanyKomunikat := sWyslanyKomunikatDummy);
					sDane := '';
				END_IF		
			END_IF
			//THD prądu, fazowe
			IF fnKomunikatDaneSzukajWartosci(sKomunikat , 'AMPERTHDL1=') = '?' OR fnKomunikatDaneSzukajWartosci(sKomunikat , 'ALL=') = '?' THEN
				fnKomunikatDaneDodaj_xOverFlow(sDane := sDane , sAtrybut := 'AMPERTHDL1=' , sWartosc := REAL_TO_STRING(rTHDPraduL1) , xOverFlow := xOverFlow);	
				IF xOverFlow = TRUE THEN
					fnZapiszKomunikat(	sCalyKomunikat := '' ,
								sTypKomunikatu := 'A' ,
								sMnemonik := sMnemonik ,
								sMACAdres := sMACAdres ,
								sIDNadawcy := sIdInstancji ,
								sIDOdbiorcy := sIdAplikacji ,
								sDaneZapasowe := sDaneZapasowe ,
								sDane := sDane ,
								arTablicaKomunikatow := arTablicaKomunikatow ,
								intTablicaKomunikatowZnacznikZapisu := intTablicaKomunikatowZnacznikZapisu ,
								intTablicaKomunikatowRozmiar := intTablicaKomunikatowRozmiar ,
								sWyslanyKomunikat := sWyslanyKomunikatDummy);
					sDane := '';
				END_IF	
			END_IF
			IF fnKomunikatDaneSzukajWartosci(sKomunikat , 'AMPERTHDL2=') = '?' OR fnKomunikatDaneSzukajWartosci(sKomunikat , 'ALL=') = '?' THEN
				fnKomunikatDaneDodaj_xOverFlow(sDane := sDane , sAtrybut := 'AMPERTHDL2=' , sWartosc := REAL_TO_STRING(rTHDPraduL2) , xOverFlow := xOverFlow);	
				IF xOverFlow = TRUE THEN
					fnZapiszKomunikat(	sCalyKomunikat := '' ,
								sTypKomunikatu := 'A' ,
								sMnemonik := sMnemonik ,
								sMACAdres := sMACAdres ,
								sIDNadawcy := sIdInstancji ,
								sIDOdbiorcy := sIdAplikacji ,
								sDaneZapasowe := sDaneZapasowe ,
								sDane := sDane ,
								arTablicaKomunikatow := arTablicaKomunikatow ,
								intTablicaKomunikatowZnacznikZapisu := intTablicaKomunikatowZnacznikZapisu ,
								intTablicaKomunikatowRozmiar := intTablicaKomunikatowRozmiar ,
								sWyslanyKomunikat := sWyslanyKomunikatDummy);
					sDane := '';
				END_IF	
			END_IF	
			IF fnKomunikatDaneSzukajWartosci(sKomunikat , 'AMPERTHDL3=') = '?' OR fnKomunikatDaneSzukajWartosci(sKomunikat , 'ALL=') = '?' THEN
				fnKomunikatDaneDodaj_xOverFlow(sDane := sDane , sAtrybut := 'AMPERTHDL3=' , sWartosc := REAL_TO_STRING(rTHDPraduL3) , xOverFlow := xOverFlow);	
				IF xOverFlow = TRUE THEN
					fnZapiszKomunikat(	sCalyKomunikat := '' ,
								sTypKomunikatu := 'A' ,
								sMnemonik := sMnemonik ,
								sMACAdres := sMACAdres ,
								sIDNadawcy := sIdInstancji ,
								sIDOdbiorcy := sIdAplikacji ,
								sDaneZapasowe := sDaneZapasowe ,
								sDane := sDane ,
								arTablicaKomunikatow := arTablicaKomunikatow ,
								intTablicaKomunikatowZnacznikZapisu := intTablicaKomunikatowZnacznikZapisu ,
								intTablicaKomunikatowRozmiar := intTablicaKomunikatowRozmiar ,
								sWyslanyKomunikat := sWyslanyKomunikatDummy);
					sDane := '';
				END_IF	
			END_IF
			
			//pytanie o stany alarmów
			IF fnKomunikatDaneSzukajWartosci(sKomunikat , 'ALARM=') = '?' OR fnKomunikatDaneSzukajWartosci(sKomunikat , 'ALL=') = '?' THEN
				FOR intPetla := 1 TO 20 BY 1 DO
					//raportowanie typu E (stanów alarmów) na zapytanie typu Q
					IF arErrorStan[intPetla] <> enumAlarmWartosc.StanNieznany THEN
						fnZapiszKomunikat(	sCalyKomunikat := '' ,
											sTypKomunikatu := 'E' ,
											sMnemonik := sMnemonik ,
											sMACAdres := sMACAdres ,
											sIDNadawcy := sIdInstancji ,
											sIDOdbiorcy := sIdAplikacji ,
											sDaneZapasowe := sDaneZapasowe ,
											sDane := fnKomunikatDaneErrorRetry(xAktywny := arErrorStan[intPetla] = enumAlarmWartosc.StanAlarmowy , intKlasa := arErrorKlasa[intPetla] , intNumer := intPetla),
											arTablicaKomunikatow := arTablicaKomunikatow ,
											intTablicaKomunikatowZnacznikZapisu := intTablicaKomunikatowZnacznikZapisu ,
											intTablicaKomunikatowRozmiar := intTablicaKomunikatowRozmiar ,
											sWyslanyKomunikat := sWyslanyKomunikatDummy);
					END_IF
				END_FOR
			END_IF
		END_IF
		//raportowanie typu A na zapytanie Q
		IF sDane <> '' THEN
			fnZapiszKomunikat(	sCalyKomunikat := '' ,
								sTypKomunikatu := 'A' ,
								sMnemonik := sMnemonik ,
								sMACAdres := sMACAdres ,
								sIDNadawcy := sIdInstancji ,
								sIDOdbiorcy := sIdAplikacji ,
								sDaneZapasowe := sDaneZapasowe ,
								sDane := sDane ,
								arTablicaKomunikatow := arTablicaKomunikatow ,
								intTablicaKomunikatowZnacznikZapisu := intTablicaKomunikatowZnacznikZapisu ,
								intTablicaKomunikatowRozmiar := intTablicaKomunikatowRozmiar ,
								sWyslanyKomunikat := sWyslanyKomunikatDummy);
		END_IF
	END_IF
END_IF

// dokonywanie obliczeń
	// Napięcia fazowe
fbNapiecieL1(	rWartoscWejsciowa := DINT_TO_REAL(SHL(wNapiecieL1Hi, 16) OR wNapiecieL1Lo), 
				rWartoscWejsciowaZaraportowana := rNapiecieL1Zaraportowana,
				rDeadband := 5,
				tCzasMinimalny := tMinimalnyCzasRaportowania,
				tCzasMaksymalny := tMaksymalnyCzasRaportowania,
				rWynikMnoznik := 0.01,
				rWartoscWyjsciowa => rNapiecieL1);

fbNapiecieL2(	rWartoscWejsciowa := DINT_TO_REAL(SHL(wNapiecieL2Hi, 16) OR wNapiecieL2Lo),
				rWartoscWejsciowaZaraportowana := rNapiecieL2Zaraportowana,
				rDeadband := 5,
				tCzasMinimalny := tMinimalnyCzasRaportowania,
				tCzasMaksymalny := tMaksymalnyCzasRaportowania,
				rWynikMnoznik := 0.01,
				rWartoscWyjsciowa => rNapiecieL2);

fbNapiecieL3(	rWartoscWejsciowa := DINT_TO_REAL(SHL(wNapiecieL3Hi, 16) OR wNapiecieL3Lo),
				rWartoscWejsciowaZaraportowana := rNapiecieL3Zaraportowana,
				rDeadband := 5,
				tCzasMinimalny := tMinimalnyCzasRaportowania,
				tCzasMaksymalny := tMaksymalnyCzasRaportowania,
				rWynikMnoznik := 0.01,
				rWartoscWyjsciowa => rNapiecieL3);
				
	// Napięcia przewodowe
fbNapiecieL1L2(	rWartoscWejsciowa := DINT_TO_REAL(SHL(wNapiecieL1L2Hi, 16) OR wNapiecieL1L2Lo),
				rWartoscWejsciowaZaraportowana := rNapiecieL1L2Zaraportowana,
				rDeadband := 3,
				tCzasMinimalny := tMinimalnyCzasRaportowania,
				tCzasMaksymalny := tMaksymalnyCzasRaportowania,
				rWynikMnoznik := 0.01,
				rWartoscWyjsciowa => rNapiecieL1L2);

fbNapiecieL2L3(	rWartoscWejsciowa := DINT_TO_REAL(SHL(wNapiecieL2L3Hi, 16) OR wNapiecieL2L3Lo),
				rWartoscWejsciowaZaraportowana := rNapiecieL2L3Zaraportowana,
				rDeadband := 3,
				tCzasMinimalny := tMinimalnyCzasRaportowania,
				tCzasMaksymalny := tMaksymalnyCzasRaportowania,
				rWynikMnoznik := 0.01,
				rWartoscWyjsciowa => rNapiecieL2L3);

fbNapiecieL3L1(	rWartoscWejsciowa := DINT_TO_REAL(SHL(wNapiecieL3L1Hi, 16) OR wNapiecieL3L1Lo),
				rWartoscWejsciowaZaraportowana := rNapiecieL3L1Zaraportowana,
				rDeadband := 3,
				tCzasMinimalny := tMinimalnyCzasRaportowania,
				tCzasMaksymalny := tMaksymalnyCzasRaportowania,
				rWynikMnoznik := 0.01,
				rWartoscWyjsciowa => rNapiecieL3L1);
				
	// Częstotliwość
fbCzestotliwosc(	rWartoscWejsciowa := DINT_TO_REAL(SHL(wCzestotliwoscHi, 16) OR wCzestotliwoscLo),
					rWartoscWejsciowaZaraportowana := rCzestotliwoscZaraportowana,
					rDeadband := 0.05,
					tCzasMinimalny := tMinimalnyCzasRaportowania,
					tCzasMaksymalny := tMaksymalnyCzasRaportowania,
					rWynikMnoznik := 0.01,
					rWartoscWyjsciowa => rCzestotliwosc);
				
	// Czas pracy
fbCzasPracyAnalizatora(	rWartoscWejsciowa := DINT_TO_REAL(SHL(wCzasPracyAnalizatoraHi, 16) OR wCzasPracyAnalizatoraLo),
						rWartoscWejsciowaZaraportowana := rCzasPracyAnalizatoraZaraportowana,
						rDeadband := 1,
						tCzasMinimalny := tMaksymalnyCzasRaportowania,
						tCzasMaksymalny := tMaksymalnyCzasRaportowania,
						rWynikMnoznik := 36,
						rWartoscWyjsciowa => rCzasPracyAnalizatora);
				
	// Prądy fazowe
fbPradL1(	rWartoscWejsciowa := DINT_TO_REAL(SHL(wPradL1Hi, 16) OR wPradL1Lo),
			rWartoscWejsciowaZaraportowana := rPradL1Zaraportowana,
			rDeadband := 3,
			tCzasMinimalny := tMinimalnyCzasRaportowania,
			tCzasMaksymalny := tMaksymalnyCzasRaportowania,
			rWynikMnoznik := 0.001,
			rWartoscWyjsciowa => rPradL1);

fbPradL2(	rWartoscWejsciowa := DINT_TO_REAL(SHL(wPradL2Hi, 16) OR wPradL2Lo),
			rWartoscWejsciowaZaraportowana := rPradL2Zaraportowana,
			rDeadband := 3,
			tCzasMinimalny := tMinimalnyCzasRaportowania,
			tCzasMaksymalny := tMaksymalnyCzasRaportowania,
			rWynikMnoznik := 0.001,
			rWartoscWyjsciowa => rPradL2);

fbPradL3(	rWartoscWejsciowa := DINT_TO_REAL(SHL(wPradL3Hi, 16) OR wPradL3Lo),
			rWartoscWejsciowaZaraportowana := rPradL3Zaraportowana,
			rDeadband := 3,
			tCzasMinimalny := tMinimalnyCzasRaportowania,
			tCzasMaksymalny := tMaksymalnyCzasRaportowania,
			rWynikMnoznik := 0.001,
			rWartoscWyjsciowa => rPradL3);

fbPradN(	rWartoscWejsciowa := DINT_TO_REAL(SHL(wPradNHi, 16) OR wPradNLo),
			rWartoscWejsciowaZaraportowana := rPradNZaraportowana,
			rDeadband := 3,
			tCzasMinimalny := tMinimalnyCzasRaportowania,
			tCzasMaksymalny := tMaksymalnyCzasRaportowania,
			rWynikMnoznik := 0.001,
			rWartoscWyjsciowa => rPradN);
				
	// Prądy średnie fazowe
fbPradSredniL1(	rWartoscWejsciowa := DINT_TO_REAL(SHL(wPradSredniL1Hi, 16) OR wPradSredniL1Lo),
				rWartoscWejsciowaZaraportowana := rPradSredniL1Zaraportowana,
				rDeadband := 1.5,
				tCzasMinimalny := tMinimalnyCzasRaportowania,
				tCzasMaksymalny := tMaksymalnyCzasRaportowania,
				rWynikMnoznik := 0.001,
				rWartoscWyjsciowa => rPradSredniL1);

fbPradSredniL2(	rWartoscWejsciowa := DINT_TO_REAL(SHL(wPradSredniL2Hi, 16) OR wPradSredniL2Lo),
				rWartoscWejsciowaZaraportowana := rPradSredniL2Zaraportowana,
				rDeadband := 1.5,
				tCzasMinimalny := tMinimalnyCzasRaportowania,
				tCzasMaksymalny := tMaksymalnyCzasRaportowania,
				rWynikMnoznik := 0.001,
				rWartoscWyjsciowa => rPradSredniL2);

fbPradSredniL3(	rWartoscWejsciowa := DINT_TO_REAL(SHL(wPradSredniL3Hi, 16) OR wPradSredniL3Lo),
				rWartoscWejsciowaZaraportowana := rPradSredniL3Zaraportowana,
				rDeadband := 1.5,
				tCzasMinimalny := tMinimalnyCzasRaportowania,
				tCzasMaksymalny := tMaksymalnyCzasRaportowania,
				rWynikMnoznik := 0.001,
				rWartoscWyjsciowa => rPradSredniL3);
				
	// Prąd średni (I1+I2+I3)/3
fbPradSredni(	rWartoscWejsciowa := (rPradSredniL1 + rPradSredniL2 + rPradSredniL3) / 3,
				rWartoscWejsciowaZaraportowana := rPradSredniZaraportowana,
				rDeadband := 1.5,
				tCzasMinimalny := tMinimalnyCzasRaportowania,
				tCzasMaksymalny := tMaksymalnyCzasRaportowania,
				rWynikMnoznik := 1,
				rWartoscWyjsciowa => rPradSredni);
				
	// Moce 3-fazowe
fbMocCzynnaCalkowita(	rWartoscWejsciowa := DINT_TO_REAL(SHL(wMocCzynnaCalkowitaHi, 16) OR wMocCzynnaCalkowitaLo),
						rWartoscWejsciowaZaraportowana := rMocCzynnaCalkowitaZaraportowana,
						rDeadband := 1000,
						tCzasMinimalny := tMinimalnyCzasRaportowania,
						tCzasMaksymalny := tMaksymalnyCzasRaportowania,
						rWynikMnoznik := 10,
						rWartoscWyjsciowa => rMocCzynnaCalkowita);
	
fbMocBiernaCalkowita(	rWartoscWejsciowa := DINT_TO_REAL(SHL(wMocBiernaCalkowitaHi, 16) OR wMocBiernaCalkowitaLo),
						rWartoscWejsciowaZaraportowana := rMocBiernaCalkowitaZaraportowana,
						rDeadband := 100,
						tCzasMinimalny := tMinimalnyCzasRaportowania,
						tCzasMaksymalny := tMaksymalnyCzasRaportowania,
						rWynikMnoznik := 10,
						rWartoscWyjsciowa => rMocBiernaCalkowita);

fbMocPozornaCalkowita(	rWartoscWejsciowa := DINT_TO_REAL(SHL(wMocPozornaCalkowitaHi, 16) OR wMocPozornaCalkowitaLo),
						rWartoscWejsciowaZaraportowana := rMocPozornaCalkowitaZaraportowana,
						rDeadband := 1000,
						tCzasMinimalny := tMinimalnyCzasRaportowania,
						tCzasMaksymalny := tMaksymalnyCzasRaportowania,
						rWynikMnoznik := 10,
						rWartoscWyjsciowa => rMocPozornaCalkowita);
		
	// Całkowity współczynnik mocy
fbWspolczynnikMocyCalkowity(	rWartoscWejsciowa := DINT_TO_REAL(SHL(wWspolczynnikMocyCalkowityHi, 16) OR wWspolczynnikMocyCalkowityLo),
								rWartoscWejsciowaZaraportowana := rWspolczynnikMocyCalkowityZaraportowana,
								rDeadband := 0.05,
								tCzasMinimalny := tMinimalnyCzasRaportowania,
								tCzasMaksymalny := tMaksymalnyCzasRaportowania,
								rWynikMnoznik := 0.001,
								rWartoscWyjsciowa => rWspolczynnikMocyCalkowity);
				
	// Moce czynne fazowe
fbMocCzynnaL1(	rWartoscWejsciowa := DINT_TO_REAL(SHL(wMocCzynnaL1Hi, 16) OR wMocCzynnaL1Lo),
				rWartoscWejsciowaZaraportowana := rMocCzynnaL1Zaraportowana,
				rDeadband := 500,
				tCzasMinimalny := tMinimalnyCzasRaportowania,
				tCzasMaksymalny := tMaksymalnyCzasRaportowania,
				rWynikMnoznik := 10,
				rWartoscWyjsciowa => rMocCzynnaL1);
				
fbMocCzynnaL2(	rWartoscWejsciowa := DINT_TO_REAL(SHL(wMocCzynnaL2Hi, 16) OR wMocCzynnaL2Lo),
				rWartoscWejsciowaZaraportowana := rMocCzynnaL2Zaraportowana,
				rDeadband := 500,
				tCzasMinimalny := tMinimalnyCzasRaportowania,
				tCzasMaksymalny := tMaksymalnyCzasRaportowania,
				rWynikMnoznik := 10,
				rWartoscWyjsciowa => rMocCzynnaL2);
				
fbMocCzynnaL3(	rWartoscWejsciowa := DINT_TO_REAL(SHL(wMocCzynnaL3Hi, 16) OR wMocCzynnaL3Lo),
				rWartoscWejsciowaZaraportowana := rMocCzynnaL3Zaraportowana,
				rDeadband := 500,
				tCzasMinimalny := tMinimalnyCzasRaportowania,
				tCzasMaksymalny := tMaksymalnyCzasRaportowania,
				rWynikMnoznik := 10,
				rWartoscWyjsciowa => rMocCzynnaL3);

	// Moce bierne fazowe
fbMocBiernaL1(	rWartoscWejsciowa := DINT_TO_REAL(SHL(wMocBiernaL1Hi, 16) OR wMocBiernaL1Lo),
				rWartoscWejsciowaZaraportowana := rMocBiernaL1Zaraportowana,
				rDeadband := 50,
				tCzasMinimalny := tMinimalnyCzasRaportowania,
				tCzasMaksymalny := tMaksymalnyCzasRaportowania,
				rWynikMnoznik := 10,
				rWartoscWyjsciowa => rMocBiernaL1);
				
fbMocBiernaL2(	rWartoscWejsciowa := DINT_TO_REAL(SHL(wMocBiernaL2Hi, 16) OR wMocBiernaL2Lo),
				rWartoscWejsciowaZaraportowana := rMocBiernaL2Zaraportowana,
				rDeadband := 50,
				tCzasMinimalny := tMinimalnyCzasRaportowania,
				tCzasMaksymalny := tMaksymalnyCzasRaportowania,
				rWynikMnoznik := 10,
				rWartoscWyjsciowa => rMocBiernaL2);
				
fbMocBiernaL3(	rWartoscWejsciowa := DINT_TO_REAL(SHL(wMocBiernaL3Hi, 16) OR wMocBiernaL3Lo),
				rWartoscWejsciowaZaraportowana := rMocBiernaL3Zaraportowana,
				rDeadband := 50,sdfgsdfg
				tCzasMinimalny := tMinimalnyCzasRaportowania,
				tCzasMaksymalny := tMaksymalnyCzasRaportowania,
				rWynikMnoznik := 10,
				rWartoscWyjsciowa => rMocBiernaL3);
				
	// Moce pozorne fazowe
fbMocPozornaL1(	rWartoscWejsciowa := DINT_TO_REAL(SHL(wMocPozornaL1Hi, 16) OR wMocPozornaL1Lo),
				rWartoscWejsciowaZaraportowana := rMocPozornaL1Zaraportowana,
				rDeadband := 500,
				tCzasMinimalny := tMinimalnyCzasRaportowania,
				tCzasMaksymalny := tMaksymalnyCzasRaportowania,
				rWynikMnoznik := 10,
				rWartoscWyjsciowa => rMocPozornaL1);
				
fbMocPozornaL2(	rWartoscWejsciowa := DINT_TO_REAL(SHL(wMocPozornaL2Hi, 16) OR wMocPozornaL2Lo),
				rWartoscWejsciowaZaraportowana := rMocPozornaL2Zaraportowana,
				rDeadband := 500,
				tCzasMinimalny := tMinimalnyCzasRaportowania,
				tCzasMaksymalny := tMaksymalnyCzasRaportowania,
				rWynikMnoznik := 10,
				rWartoscWyjsciowa => rMocPozornaL2);
				
fbMocPozornaL3(	rWartoscWejsciowa := DINT_TO_REAL(SHL(wMocPozornaL3Hi, 16) OR wMocPozornaL3Lo),
				rWartoscWejsciowaZaraportowana := rMocPozornaL3Zaraportowana,
				rDeadband := 500,
				tCzasMinimalny := tMinimalnyCzasRaportowania,
				tCzasMaksymalny := tMaksymalnyCzasRaportowania,
				rWynikMnoznik := 10,
				rWartoscWyjsciowa => rMocPozornaL3);
				
	// Współczynniki mocy fazowe
fbWspolczynnikMocyL1(	rWartoscWejsciowa := DINT_TO_REAL(SHL(wWspolczynnikMocyL1Hi, 16) OR wWspolczynnikMocyL1Lo),
						rWartoscWejsciowaZaraportowana := rWspolczynnikMocyL1Zaraportowana,
						rDeadband := 0.05,
						tCzasMinimalny := tMinimalnyCzasRaportowania,
						tCzasMaksymalny := tMaksymalnyCzasRaportowania,
						rWynikMnoznik := 0.001,
						rWartoscWyjsciowa => rWspolczynnikMocyL1);
				
fbWspolczynnikMocyL2(	rWartoscWejsciowa := DINT_TO_REAL(SHL(wWspolczynnikMocyL2Hi, 16) OR wWspolczynnikMocyL2Lo),
						rWartoscWejsciowaZaraportowana := rWspolczynnikMocyL2Zaraportowana,
						rDeadband := 0.05,
						tCzasMinimalny := tMinimalnyCzasRaportowania,
						tCzasMaksymalny := tMaksymalnyCzasRaportowania,
						rWynikMnoznik := 0.001,
						rWartoscWyjsciowa => rWspolczynnikMocyL2);
				
fbWspolczynnikMocyL3(	rWartoscWejsciowa := DINT_TO_REAL(SHL(wWspolczynnikMocyL3Hi, 16) OR wWspolczynnikMocyL3Lo),
						rWartoscWejsciowaZaraportowana := rWspolczynnikMocyL3Zaraportowana,
						rDeadband := 0.05,
						tCzasMinimalny := tMinimalnyCzasRaportowania,
						tCzasMaksymalny := tMaksymalnyCzasRaportowania,
						rWynikMnoznik := 0.001,
						rWartoscWyjsciowa => rWspolczynnikMocyL3);
				
	// Energia pobrana
fbEnergiaCzynnaPobrana(	rWartoscWejsciowa := DINT_TO_REAL(SHL(wEnergiaCzynnaPobranaHi, 16) OR wEnergiaCzynnaPobranaLo),
						rWartoscWejsciowaZaraportowana := rEnergiaCzynnaPobranaZaraportowana,
						rDeadband := 3600000,
						tCzasMinimalny := tMinimalnyCzasRaportowania,
						tCzasMaksymalny := tMaksymalnyCzasRaportowania,
						rWynikMnoznik := 3600000,
						rWartoscWyjsciowa => rEnergiaCzynnaPobrana);
				
fbEnergiaBiernaPobrana(	rWartoscWejsciowa := DINT_TO_REAL(SHL(wEnergiaBiernaPobranaHi, 16) OR wEnergiaBiernaPobranaLo),
						rWartoscWejsciowaZaraportowana := rEnergiaBiernaPobranaZaraportowana,
						rDeadband := 1800000,
						tCzasMinimalny := tMinimalnyCzasRaportowania,
						tCzasMaksymalny := tMaksymalnyCzasRaportowania,
						rWynikMnoznik := 3600000,
						rWartoscWyjsciowa => rEnergiaBiernaPobrana);
				
fbEnergiaPozornaPobrana(	rWartoscWejsciowa := DINT_TO_REAL(SHL(wEnergiaPozornaPobranaHi, 16) OR wEnergiaPozornaPobranaLo),
							rWartoscWejsciowaZaraportowana := rEnergiaPozornaPobranaZaraportowana,
							rDeadband := 3600000,
							tCzasMinimalny := tMinimalnyCzasRaportowania,
							tCzasMaksymalny := tMaksymalnyCzasRaportowania,
							rWynikMnoznik := 3600000,
							rWartoscWyjsciowa => rEnergiaPozornaPobrana);

	// Moce średnie
fbMocCzynnaSrednia(	rWartoscWejsciowa := DINT_TO_REAL(SHL(wMocCzynnaSredniaHi, 16) OR wMocCzynnaSredniaLo),
					rWartoscWejsciowaZaraportowana := rMocCzynnaSredniaZaraportowana,
					rDeadband := 500,
					tCzasMinimalny := tMinimalnyCzasRaportowania,
					tCzasMaksymalny := tMaksymalnyCzasRaportowania,
					rWynikMnoznik := 10,
					rWartoscWyjsciowa => rMocCzynnaSrednia);
				
fbMocBiernaSrednia(	rWartoscWejsciowa := DINT_TO_REAL(SHL(wMocBiernaSredniaHi, 16) OR wMocBiernaSredniaLo),
					rWartoscWejsciowaZaraportowana := rMocBiernaSredniaZaraportowana,
					rDeadband := 500,
					tCzasMinimalny := tMinimalnyCzasRaportowania,
					tCzasMaksymalny := tMaksymalnyCzasRaportowania,
					rWynikMnoznik := 10,
					rWartoscWyjsciowa => rMocBiernaSrednia);
				
fbMocPozornaSrednia(	rWartoscWejsciowa := DINT_TO_REAL(SHL(wMocPozornaSredniaHi, 16) OR wMocPozornaSredniaLo),
						rWartoscWejsciowaZaraportowana := rMocPozornaSredniaZaraportowana,
						rDeadband := 500,
						tCzasMinimalny := tMinimalnyCzasRaportowania,
						tCzasMaksymalny := tMaksymalnyCzasRaportowania,
						rWynikMnoznik := 10,
						rWartoscWyjsciowa => rMocPozornaSrednia);
				
	//Maksymalne napięcia fazowe
fbMaksymalneNapiecieL1(	rWartoscWejsciowa := DINT_TO_REAL(SHL(wMaksymalneNapiecieL1Hi, 16) OR wMaksymalneNapiecieL1Lo),
				rWartoscWejsciowaZaraportowana := rMaksymalneNapiecieL1Zaraportowana,
				rDeadband := 20,
				tCzasMinimalny := tMinimalnyCzasRaportowania,
				tCzasMaksymalny := tMaksymalnyCzasRaportowania,
				rWynikMnoznik := 0.01,
				rWartoscWyjsciowa => rMaksymalneNapiecieL1);
				
fbMaksymalneNapiecieL2(	rWartoscWejsciowa := DINT_TO_REAL(SHL(wMaksymalneNapiecieL2Hi, 16) OR wMaksymalneNapiecieL2Lo),
				rWartoscWejsciowaZaraportowana := rMaksymalneNapiecieL2Zaraportowana,
				rDeadband := 20,
				tCzasMinimalny := tMinimalnyCzasRaportowania,
				tCzasMaksymalny := tMaksymalnyCzasRaportowania,
				rWynikMnoznik := 0.01,
				rWartoscWyjsciowa => rMaksymalneNapiecieL2);
				
fbMaksymalneNapiecieL3(	rWartoscWejsciowa := DINT_TO_REAL(SHL(wMaksymalneNapiecieL3Hi, 16) OR wMaksymalneNapiecieL3Lo),
				rWartoscWejsciowaZaraportowana := rMaksymalneNapiecieL3Zaraportowana,
				rDeadband := 20,
				tCzasMinimalny := tMinimalnyCzasRaportowania,
				tCzasMaksymalny := tMaksymalnyCzasRaportowania,
				rWynikMnoznik := 0.01,
				rWartoscWyjsciowa => rMaksymalneNapiecieL3);
			
	// THD napięcia
fbTHDNapieciaL1(	rWartoscWejsciowa := WORD_TO_REAL(wTHDNapieciaL1),
					rWartoscWejsciowaZaraportowana := rTHDNapieciaL1Zaraportowana,
					rDeadband := 0.08,
					tCzasMinimalny := tMinimalnyCzasRaportowania,
					tCzasMaksymalny := tMaksymalnyCzasRaportowania,
					rWynikMnoznik := 0.001,
					rWartoscWyjsciowa => rTHDNapieciaL1);
				
fbTHDNapieciaL2(	rWartoscWejsciowa := WORD_TO_REAL(wTHDNapieciaL2),
					rWartoscWejsciowaZaraportowana := rTHDNapieciaL2Zaraportowana,
					rDeadband := 0.08,
					tCzasMinimalny := tMinimalnyCzasRaportowania,
					tCzasMaksymalny := tMaksymalnyCzasRaportowania,
					rWynikMnoznik := 0.001,
					rWartoscWyjsciowa => rTHDNapieciaL2);
				
fbTHDNapieciaL3(	rWartoscWejsciowa := WORD_TO_REAL(wTHDNapieciaL3),
					rWartoscWejsciowaZaraportowana := rTHDNapieciaL3Zaraportowana,
					rDeadband := 0.08,
					tCzasMinimalny := tMinimalnyCzasRaportowania,
					tCzasMaksymalny := tMaksymalnyCzasRaportowania,
					rWynikMnoznik := 0.001,
					rWartoscWyjsciowa => rTHDNapieciaL3);
				
	// THD prądu
fbTHDPraduL1(	rWartoscWejsciowa := WORD_TO_REAL(wTHDPraduL1),
				rWartoscWejsciowaZaraportowana := rTHDPraduL1Zaraportowana,
				rDeadband := 0.08,
				tCzasMinimalny := tMinimalnyCzasRaportowania,
				tCzasMaksymalny := tMaksymalnyCzasRaportowania,
				rWynikMnoznik := 0.001,
				rWartoscWyjsciowa => rTHDPraduL1);
				
fbTHDPraduL2(	rWartoscWejsciowa := WORD_TO_REAL(wTHDPraduL2),
				rWartoscWejsciowaZaraportowana := rTHDPraduL2Zaraportowana,
				rDeadband := 0.08,
				tCzasMinimalny := tMinimalnyCzasRaportowania,
				tCzasMaksymalny := tMaksymalnyCzasRaportowania,
				rWynikMnoznik := 0.001,
				rWartoscWyjsciowa => rTHDPraduL2);
				
fbTHDPraduL3(	rWartoscWejsciowa := WORD_TO_REAL(wTHDPraduL3),
				rWartoscWejsciowaZaraportowana := rTHDPraduL3Zaraportowana,
				rDeadband := 0.08,
				tCzasMinimalny := tMinimalnyCzasRaportowania,
				tCzasMaksymalny := tMaksymalnyCzasRaportowania,
				rWynikMnoznik := 0.001,
				rWartoscWyjsciowa => rTHDPraduL3);
				
	
//Raportowanie typu M do IZE wartosci odczytanych z Modbusa			
IF (rNapiecieL1 <> rNapiecieL1Zaraportowana OR rNapiecieL2 <> rNapiecieL2Zaraportowana OR rNapiecieL3 <> rNapiecieL3Zaraportowana OR rNapiecieL1L2 <> rNapiecieL1L2Zaraportowana 
OR rNapiecieL2L3 <> rNapiecieL2L3Zaraportowana OR rNapiecieL3L1 <> rNapiecieL3L1Zaraportowana OR rCzestotliwosc <> rCzestotliwoscZaraportowana OR rCzasPracyAnalizatora <> rCzasPracyAnalizatoraZaraportowana 
OR rPradL1 <> rPradL1Zaraportowana OR rPradL2 <> rPradL2Zaraportowana OR rPradL3 <> rPradL3Zaraportowana OR rPradN <> rPradNZaraportowana OR rPradSredniL1 <> rPradSredniL1Zaraportowana 
OR rPradSredniL2 <> rPradSredniL2Zaraportowana OR rPradSredniL3 <> rPradSredniL3Zaraportowana OR rPradSredni <> rPradSredniZaraportowana OR rMocCzynnaCalkowita <> rMocCzynnaCalkowitaZaraportowana 
OR rMocBiernaCalkowita <> rMocBiernaCalkowitaZaraportowana OR rMocPozornaCalkowita <> rMocPozornaCalkowitaZaraportowana OR rWspolczynnikMocyCalkowity <> rWspolczynnikMocyCalkowityZaraportowana 
OR rMocCzynnaL1 <> rMocCzynnaL1Zaraportowana OR rMocCzynnaL2 <> rMocCzynnaL2Zaraportowana OR rMocCzynnaL3 <> rMocCzynnaL3Zaraportowana OR rMocBiernaL1 <> rMocBiernaL1Zaraportowana 
OR rMocBiernaL2 <> rMocBiernaL2Zaraportowana OR rMocBiernaL3 <> rMocBiernaL3Zaraportowana OR rMocPozornaL1 <> rMocPozornaL1Zaraportowana OR rMocPozornaL2 <> rMocPozornaL2Zaraportowana 
OR rMocPozornaL3 <> rMocPozornaL3Zaraportowana OR rWspolczynnikMocyL1 <> rWspolczynnikMocyL1Zaraportowana OR rWspolczynnikMocyL2 <> rWspolczynnikMocyL2Zaraportowana 
OR rWspolczynnikMocyL3 <> rWspolczynnikMocyL3Zaraportowana OR rEnergiaCzynnaPobrana <> rEnergiaCzynnaPobranaZaraportowana OR rEnergiaBiernaPobrana <> rEnergiaBiernaPobranaZaraportowana 
OR rEnergiaPozornaPobrana <> rEnergiaPozornaPobranaZaraportowana OR rMocCzynnaSrednia <> rMocCzynnaSredniaZaraportowana OR rMocBiernaSrednia <> rMocBiernaSredniaZaraportowana 
OR rMocPozornaSrednia <> rMocPozornaSredniaZaraportowana OR rMaksymalneNapiecieL1 <> rMaksymalneNapiecieL1Zaraportowana OR rMaksymalneNapiecieL2 <> rMaksymalneNapiecieL2Zaraportowana 
OR rMaksymalneNapiecieL3 <> rMaksymalneNapiecieL3Zaraportowana OR rTHDNapieciaL1 <> rTHDNapieciaL1Zaraportowana OR rTHDNapieciaL2 <> rTHDNapieciaL2Zaraportowana OR rTHDNapieciaL3 <> rTHDNapieciaL3Zaraportowana 
OR rTHDPraduL1 <> rTHDPraduL1Zaraportowana OR rTHDPraduL2 <> rTHDPraduL2Zaraportowana OR rTHDPraduL3 <> rTHDPraduL3Zaraportowana) AND arModbusStatusKomunikacji[bAdres] = enumModbusStatus.KomunikacjaPrawidlowa 
AND xPoInicjalizacji THEN
	xRaport := TRUE;
END_IF 
				
